// TwinCAT 3 PLC project TE1063
// ProgramVersion: 3.1.4024.0
// libraries:
//   CmpBitmapPool, * (System)
//   Tc2_Database, * (Beckhoff Automation GmbH)
//   Tc2_Math, * (Beckhoff Automation GmbH)
//   Tc2_MC2, * (Beckhoff Automation GmbH)
//   Tc2_SerialCom, * (Beckhoff Automation GmbH)
//   Tc2_Standard, * (Beckhoff Automation GmbH)
//   Tc2_System, * (Beckhoff Automation GmbH)
//   Tc2_TcpIp, * (Beckhoff Automation GmbH)
//   Tc2_Utilities, * (Beckhoff Automation GmbH)
//   Tc3_EventLogger, * (Beckhoff Automation GmbH)
//   Tc3_JsonXml, * (Beckhoff Automation GmbH)
//   Tc3_Module, * (Beckhoff Automation GmbH)
//   Base Interfaces,newest,System
//   VisuSymbols,3.5.10.0,System
// project tree:
//   DUTs/AlarmEventLogger/ E_Events.TcDUT, ST_GeneralAlarm.TcDUT, ST_PumpError.TcDUT (not stored), ST_ValveError.TcDUT
//   DUTs/AutoCycle/ E_MachineStates.TcDUT, E_PrimeSolventState.TcDUT, E_RecoveryState.TcDUT, E_WashingState.TcDUT
//   DUTs/Calibration/ E_LeakTestState.TcDUT, E_PState.TcDUT, E_StopState.TcDUT, E_CalibrationStatus.TcDUT, E_CalibStep.TcDUT, E_ScaleCmd.TcDUT, E_SolventType.TcDUT, ST_CalibrationData.TcDUT, ST_CalibrationInfo.TcDUT, ST_CalibrationPump.TcDUT, ST_CalibrationPumpResult.TcDUT, ST_DosingResults.TcDUT, ST_LinearPumpCalibration.TcDUT, ST_LinearPumpControllDB.TcDUT, ST_ReportInfo.TcDUT, ST_ScaleReply.TcDUT
//   DUTs/HMI/ E_IconState.TcDUT, E_MachineMode.TcDUT (not stored), ST_AX8101IOInfo.TcDUT, ST_AMI8000IOInfo.TcDUT, ST_HMIAnimation.TcDUT, ST_HMIDigInputs.TcDUT, ST_HMIDigOutputs.TcDUT, ST_HMIManual.TcDUT, ST_HMIParameters.TcDUT, ST_InfoPage.TcDUT, ST_EL7062IOInfo.TcDUT, ST_MotorsJog.TcDUT, ST_Reminders.TcDUT
//   DUTs/ifmLvlSensors/ E_LevelSensorID.TcDUT, ST_KQ1000_Data.TcDUT
//   DUTs/IO/ ST_AL1333.TcDUT, ST_AX8108.TcDUT, ST_EL1809.TcDUT, ST_EL2624.TcDUT, ST_EL2809.TcDUT, ST_EL3022.TcDUT (not stored), ST_EL3058.TcDUT, ST_EL6631.TcDUT, ST_EL6910.TcDUT, ST_EL7062.TcDUT, ST_EL7062A1.TcDUT, ST_EL7062A2.TcDUT, ST_EL7211.TcDUT, ST_EP9208.TcDUT
//   DUTs/ManualControl/ E_SolenoidSet.TcDUT, ST_MotorCommand.TcDUT, ST_PumpCommand.TcDUT, ST_ValveCommand.TcDUT
//   DUTs/MotionControl/ E_ActuatorState.TcDUT, E_MotorType.TcDUT, E_PumpDirection.TcDUT (not stored), E_PumpPath.TcDUT, ST_ActuatorStatus.TcDUT, ST_AxisReadStatus.TcDUT, ST_Motor.TcDUT, ST_SolenoidSet.TcDUT
//   DUTs/Recipe/ ST_HMI_OtherParamsRow.TcDUT, ST_HMI_SolventAndTimeRow.TcDUT, ST_HMI_VolumesRow.TcDUT, ST_Recipe.TcDUT, ST_RecipeFileInfo.TcDUT, ST_RecipeInfo.TcDUT, ST_RecipeOtherParams.TcDUT, ST_RecipeSolventAndTimes.TcDUT, ST_RecipeVolumes.TcDUT
//   DUTs/Report/ ST_CalibHeaderTest.TcDUT, E_ReportType.TcDUT, ST_CompleteMethodHeader.TcDUT, ST_LinearReport.TcDUT, ST_ReportListItem.TcDUT, ST_ReportListItem_Test.TcDUT, ST_ReportPostRun.TcDUT, ST_RunEvent.TcDUT, ST_SolventInfo.TcDUT, ST_SystemSettingsReport.TcDUT, ST_VolumeLine.TcDUT
//   DUTs/Safety/ ST_SafetyInputs.TcDUT, ST_SafetyOutputs.TcDUT
//   DUTs/Settings/ ST_CalibrationSettings.TcDUT, ST_LeakTestSettings.TcDUT, ST_PumpSettings.TcDUT, ST_SolventsSettings.TcDUT
//   DUTs/UserManagement/ E_UserGroup.TcDUT, ST_User.TcDUT, ST_UserStats.TcDUT
//   DUTs/Utility/ E_PowerAction.TcDUT, E_SeqState.TcDUT
//   GVLs/ GVL_Alarms.TcGVL, GVL_Calibration.TcGVL, GVL_Constant.TcGVL, GVL_HMI.TcGVL, GVL_IO.TcGVL, GVL_Reports.TcGVL, GVL_Retain.TcGVL, GVL_Settings.TcGVL, GVL_Motion.TcGVL, GVL_Recipe.TcGVL, GVL_Safety.TcGVL, GVL_UserManagement.TcGVL
//   / PlcTask.TcTTO, Task_Events.TcTTO, Task_HMI.TcTTO, Task_Services.TcTTO, Visualization Manager.TcVMO (not stored)
//   POUs/0. Main/ MAIN_Control.TcPOU, MAIN_Events.TcPOU, MAIN_HMI.TcPOU, MAIN_Services.TcPOU
//   POUs/2. AutoCycle/Hardware Control/ FB_SetSolenoid.TcPOU, FB_SolenoidControl.TcPOU
//   POUs/2. AutoCycle/ PRG_AutoCycle.TcPOU
//   POUs/2. AutoCycle/Stages/ FB_MeteringSolvent1.TcPOU, FB_PostRun.TcPOU, FB_PrimeSolvent.TcPOU, FB_AirFlowCheck.TcPOU, FB_DryingPhase.TcPOU, FB_InitChecks.TcPOU, FB_LeakTest.TcPOU, FB_RecoveryPhase.TcPOU, FB_SealStages.TcPOU, FB_WashingPhase.TcPOU
//   POUs/3. HMI/ PRG_HMIControl.TcPOU, PRG_SaveSolvents.TcPOU, PRG_SetModulestatus.TcPOU
//   POUs/5. Calibration/ FB_BuildCalReportJson.TcPOU, FB_CalibrationManager.TcPOU, FB_SaveCalibrationReport.TcPOU, FB_SaveCalReportToFile.TcPOU, FB_ScaleDevice.TcPOU, PRG_Calibration.TcPOU
//   POUs/6. Reports/ PRG_ReportsManager.TcPOU
//   POUs/7. EventsAndAlarms/ FB_AlarmHandler.TcPOU, FB_ErrorHandler.TcPOU, FB_EventHandler.TcPOU (not stored)
//   POUs/7. EventsAndAlarms/Marco/ POU_EventTest.TcPOU, POU_FaultHandler.TcPOU, PRG_MasterSystemTime.TcPOU
//   POUs/Functions/ F_AnyAxisMoving.TcPOU, F_GetPumpPath.TcPOU, F_GetValvePosition.TcPOU, F_JarName.TcPOU, F_MonthString.TcPOU (not stored), F_ParseWeight.TcPOU, F_REAL_TO_STRING_2DEC.TcPOU, F_ROUND_REAL.TcPOU, F_sec_to_time.TcPOU, F_TwoDigits.TcPOU (not stored), F_VolumeToSteps.TcPOU, F_VolumeToSteps_Path.TcPOU, F_SqlEscapeString.TcPOU
//   POUs/1. MachineControl/ PRG_ManualControl.TcPOU, PRG_MasterControl.TcPOU, PRG_SafetyHandle.TcPOU, PRG_StoppedState.TcPOU, PRG_SystemInit.TcPOU, PRG_SystemReady.TcPOU
//   POUs/Levels/ FB_KQ1000_Parser.TcPOU, FB_LevelSensors.TcPOU, PRG_LevelHandler.TcPOU
//   POUs/MARCO/DB/ DB_Edit_Method.TcPOU, DB_Load_CompleteMethod.TcPOU, DB_Query.TcPOU, GVL_DB.TcGVL, DB_Load_SysParameters.TcPOU, DB_Create_Calibration.TcPOU
//   POUs/MARCO/DB/STs/ E_DB_QUERY_STATE.TcTLEO, E_UserMgmtEventType.TcDUT, ST_CalibrationReportHeader.TcDUT, ST_CalibrationReportLine.TcDUT, ST_CalibrationReportListItem.TcDUT, ST_Data_CUL.TcDUT (not stored), ST_Data_PCR.TcDUT, ST_Data_UHR.TcDUT, ST_DB_Solvents.TcDUT, ST_LinearMotors.TcDUT, ST_ListMethod.TcDUT, ST_Parameters_MR.TcDUT, ST_CompleteMethod.TcDUT, ST_Parameters_PCR.TcDUT, ST_PostRunReport.TcDUT, ST_Results.TcDUT (not stored), ST_Solvents.TcDUT, ST_SysParameters.TcDUT, ST_UserMgmtHistoryEvent.TcDUT, ST_VolumeData.TcDUT
//   POUs/MARCO/OLD/ GVL_Marco.TcGVL, POU_Master_Calib.TcPOU, POU_Master_Calib_1.TcPOU, POU_Master_Calib_2.TcPOU, POU_Motion.TcPOU (not stored)
//   POUs/Utilities/ FB_Blink.TcPOU (not stored), FB_DosingTest.TcPOU, FB_EventLog.TcPOU (not stored), FB_SensorScaling.TcPOU, FB_TCPClient.TcPOU, PRG_PowerManagement.TcPOU (not stored), PRG_RetainValveAngles.TcPOU (not stored), PRG_ShutdownPLC.TcPOU (not stored), PRG_SystemInfo.TcPOU (not stored), PRG_TowerAlarmLamps.TcPOU, PRG_UpdateVariablesMoving.TcPOU, PRG_UserManagementHistory.TcPOU, PRG_ValvePositionRecovery.TcPOU (not stored), PRG_ValveTest.TcPOU
//   POUs/MotionControl/ FB_AllPumpsController.TcPOU, FB_MotorWrapper.TcPOU, IF_Actuator.TcIO, PRG_AxisAssignment.TcPOU
//   POUs/4. RecipeHandle/ FB_DeleteRecipe.TcPOU, FB_ListRecipeFiles.TcPOU, FB_LoadRecipe.TcPOU, FB_RecipeHeaderHandler.TcPOU, FB_SaveRecipe.TcPOU, PRG_RecipeManager.TcPOU
//   VISUs/ GlobalTextList.TcGTLO, Visualization.TcVIS
// real-time tasks:
//   TASK Task_Control: cycle T#10ms, priority 10, ADS port 350
//   TASK Task_HMI: cycle T#100000us, priority 12, ADS port 351
//   TASK Task_Events: cycle T#250ms, priority 14, ADS port 352
//   TASK Task_Services: cycle T#1000ms, priority 16, ADS port 353
// motion (NC):
//   TASK NC-Task 1 SAF: cycle T#2ms, priority 4, ADS port 501
//   TASK NC-Task 1 SVB: cycle T#2ms, priority 6, ADS port 511
//   AXIS M1 Motor - SR Vertical (id 28)
//     General: UnitFlags=#x00000001
//     Dynamic: Acceleration=58.278, Deceleration=58.278, Jerk=174.834
//     Velo: RefSearch=0.38852, RefSync=0.38852, SlowManual=1.25, FastManual=7.5, Fast=38.852, Maximum=38.852
//     OtherSettings: AllowMotionCmdToSlave=true
//     encoder EncType=19
//       EncPara: ScaleFactorNumerator=25, ScaleFactorDenominator=20971520, MaxCount=#xffffffff
//     drive DrvType=16
//       DrvPara: MaxCount=#xffffffff, DriveControlDWord=#x00020100
//         Analog: VeloReferenz=42.7372, VeloScale=71.5255737304688, TorqueSetpointScale=10, ScaleFactorActTorque=0.1
//         TimeComp: TaskDelayCycles=1
//     controller CtrType=1
//       CtrPara: PriorControlFactor=1
//         Observer: BandWidth=20
//   AXIS M2 Motor - SC Vertical (id 6)
//     Dynamic: AccelerationMaximum=15, DecelerationMaximum=15, Acceleration=15, Deceleration=15, Jerk=2457.738
//     Velo: RefSearch=5.46164, RefSync=5.46164, SlowManual=2, FastManual=6, Fast=546.164, Maximum=546.164
//     OtherSettings: AllowMotionCmdToSlave=true, PulseDistancePos=1, PulseDistanceNeg=1
//     encoder EncType=19
//       EncPara: ScaleFactorNumerator=10, ScaleFactorDenominator=1048576, MaxCount=#xffffffff
//         TimeComp: TimeCompMode=1, EncDelayCycles=4
//     drive DrvType=16
//       DrvPara: MaxCount=#xffffffff, DriveControlDWord=#x00020100
//         Analog: VeloReferenz=600.7804, VeloScale=32, TorqueSetpointScale=10, ScaleFactorActTorque=0.1
//         TimeComp: TaskDelayCycles=1
//     controller CtrType=1
//       CtrPara: PriorControlFactor=1
//         Observer: BandWidth=20
//   AXIS M3 Motor - SC Horizontal (id 7)
//     Dynamic: Acceleration=819.246, Deceleration=819.246, Jerk=2457.738
//     Velo: RefSearch=5.46164, RefSync=5.46164, SlowManual=6, FastManual=12, Fast=546.164, Maximum=546.164
//     OtherSettings: AllowMotionCmdToSlave=true, PulseDistancePos=2, PulseDistanceNeg=2
//     encoder EncType=19
//       EncPara: ScaleFactorNumerator=10, ScaleFactorDenominator=1048576, MaxCount=#xffffffff
//     drive DrvType=16
//       DrvPara: MaxCount=#xffffffff, DriveControlDWord=#x00020100
//         Analog: VeloReferenz=600.7804, VeloScale=32, TorqueSetpointScale=10, ScaleFactorActTorque=0.1
//         TimeComp: TaskDelayCycles=1
//     controller CtrType=1
//       CtrPara: PriorControlFactor=1
//         Observer: BandWidth=20
//   AXIS M4 Motor - Valve 1 (id 1)
//     General: UnitName=°
//     Dynamic: Acceleration=15000, Deceleration=15000, Jerk=88478.5
//     Velo: RefSearch=196.61898, RefSync=196.61898, SlowManual=300, FastManual=1000, Fast=19661.898, Maximum=19661.9
//     OtherSettings: AllowMotionCmdToSlave=true, PulseDistancePos=1, PulseDistanceNeg=1
//     encoder EncType=19
//       EncPara: ScaleFactorNumerator=360, ScaleFactorDenominator=1048576, Offset=959.925842285156, MaxCount=#xffffffff, ReferenceSystem=4
//         SoftEndMaxControl: Range=7200
//     drive DrvType=16
//       DrvPara: MaxCount=#xffffffff, DriveControlDWord=#x00020100
//         Analog: VeloReferenz=21628.0878, VeloScale=32, TorqueSetpointScale=10, ScaleFactorActTorque=0.1
//         TimeComp: TaskDelayCycles=1
//     controller CtrType=1
//       CtrPara: PriorControlFactor=1
//         PosDiffControl: Range=90
//         Observer: BandWidth=20
//   AXIS M5 Motor - Valve 2 (id 2)
//     General: UnitName=°
//     Dynamic: Acceleration=15000, Deceleration=15000, Jerk=88478.5
//     Velo: RefSearch=196.61898, RefSync=196.61898, SlowManual=300, FastManual=1000, Fast=19661.898, Maximum=19661.9
//     OtherSettings: AllowMotionCmdToSlave=true, PulseDistancePos=1, PulseDistanceNeg=1
//     encoder EncType=19
//       EncPara: ScaleFactorNumerator=360, ScaleFactorDenominator=1048576, MaxCount=#xffffffff, ReferenceSystem=4
//     drive DrvType=16
//       DrvPara: MaxCount=#xffffffff, DriveControlDWord=#x00020100
//         Analog: VeloReferenz=21628.0878, VeloScale=32, TorqueSetpointScale=10, ScaleFactorActTorque=0.1
//         TimeComp: TaskDelayCycles=1
//     controller CtrType=1
//       CtrPara: PriorControlFactor=1
//         PosDiffControl: Range=90
//         Observer: BandWidth=20
//   AXIS M6 Motor - Valve 3 (id 29)
//     General: UnitName=°
//     Dynamic: Acceleration=15000, Deceleration=15000, Jerk=88478.5
//     Velo: RefSearch=196.61898, RefSync=196.61898, SlowManual=300, FastManual=1000, Fast=19661.898, Maximum=19661.9
//     OtherSettings: AllowMotionCmdToSlave=true, PulseDistancePos=1, PulseDistanceNeg=1
//     encoder EncType=19
//       EncPara: ScaleFactorNumerator=360, ScaleFactorDenominator=1048576, MaxCount=#xffffffff, ReferenceSystem=4
//     drive DrvType=16
//       DrvPara: MaxCount=#xffffffff, DriveControlDWord=#x00020100
//         Analog: VeloReferenz=21628.0878, VeloScale=32, TorqueSetpointScale=10, ScaleFactorActTorque=0.1
//         TimeComp: TaskDelayCycles=1
//     controller CtrType=1
//       CtrPara: PriorControlFactor=1
//         PosDiffControl: Range=90
//         Observer: BandWidth=20
//   AXIS M7 Motor - Valve 4 (id 4)
//     General: UnitName=°
//     Dynamic: Acceleration=15000, Deceleration=15000, Jerk=88478.5
//     Velo: RefSearch=196.61898, RefSync=196.61898, SlowManual=300, FastManual=1000, Fast=19661.898, Maximum=19661.9
//     OtherSettings: AllowMotionCmdToSlave=true, PulseDistancePos=1, PulseDistanceNeg=1
//     encoder EncType=19
//       EncPara: ScaleFactorNumerator=360, ScaleFactorDenominator=1048576, MaxCount=#xffffffff, ReferenceSystem=4
//     drive DrvType=16
//       DrvPara: MaxCount=#xffffffff, DriveControlDWord=#x00020100
//         Analog: VeloReferenz=21628.0878, VeloScale=32, TorqueSetpointScale=10, ScaleFactorActTorque=0.1
//         TimeComp: TaskDelayCycles=1
//     controller CtrType=1
//       CtrPara: PriorControlFactor=1
//         PosDiffControl: Range=90
//         Observer: BandWidth=20
//   AXIS M8 Motor - Valve 5 (id 5)
//     General: UnitName=°
//     Dynamic: Acceleration=15000, Deceleration=15000, Jerk=88478.541
//     Velo: RefSearch=196.61898, RefSync=196.61898, SlowManual=300, FastManual=1000, Fast=19661.898, Maximum=19661.898
//     OtherSettings: AllowMotionCmdToSlave=true, PulseDistancePos=1, PulseDistanceNeg=1
//     encoder EncType=19
//       EncPara: ScaleFactorNumerator=360, ScaleFactorDenominator=1048576, MaxCount=#xffffffff, ReferenceSystem=4
//     drive DrvType=16
//       DrvPara: MaxCount=#xffffffff, DriveControlDWord=#x00020100
//         Analog: VeloReferenz=21628.0878, VeloScale=32, TorqueSetpointScale=10, ScaleFactorActTorque=0.1
//         TimeComp: TaskDelayCycles=1
//     controller CtrType=1
//       CtrPara: PriorControlFactor=1
//         PosDiffControl: Range=90
//         Observer: BandWidth=20
//   AXIS Pump 1 - Linear (id 8)
//     Dynamic: Acceleration=7200, Deceleration=7200, Jerk=21600
//     Velo: RefSearch=48, RefSync=48, SlowManual=50, FastManual=100, Fast=4800, Maximum=4800
//     OtherSettings: AllowMotionCmdToSlave=true, PulseDistancePos=1, PulseDistanceNeg=1
//     encoder EncType=19
//       EncPara: ScaleFactorNumerator=200, ScaleFactorDenominator=1048576, MaxCount=#xffffffff
//         SoftEndMinControl: Range=-4500
//         SoftEndMaxControl: Range=500
//     drive DrvType=16
//       DrvPara: MaxCount=#xffffffff, DriveControlDWord=#x00020100
//         Analog: VeloReferenz=5280, VeloScale=32, TorqueSetpointScale=10, ScaleFactorActTorque=0.1
//         TimeComp: TaskDelayCycles=1
//     controller CtrType=1
//       CtrPara: PriorControlFactor=1
//         Observer: BandWidth=20
//   AXIS Pump 1 - Rotary (id 9)
//     General: UnitName=°
//     Dynamic: AccelerationMaximum=1500, DecelerationMaximum=1500, Jerk=21793.7205
//     Velo: RefSearch=48.43049, RefSync=48.43049, SlowManual=242.15245, FastManual=1452.9147, Fast=4843.049, Maximum=6000
//     OtherSettings: AllowMotionCmdToSlave=true
//     encoder EncType=19
//       EncPara: ScaleFactorNumerator=360, ScaleFactorDenominator=1048576, MaxCount=#xffffffff
//         Inc: RefSyncInverse=false
//     drive DrvType=16
//       DrvPara: MaxCount=#xffffffff, DriveControlDWord=#x00020100
//         Analog: VeloReferenz=5500, VeloScale=32, TorqueSetpointScale=10, ScaleFactorActTorque=0.1
//         TimeComp: TaskDelayCycles=1
//     controller CtrType=2
//       CtrPara: PriorControlFactor=1
//         PosDiffControl: Range=200
//         Observer: BandWidth=20
//   AXIS Pump 2 - Linear (id 10)
//     Dynamic: Acceleration=7200, Deceleration=7200, Jerk=21600
//     Velo: RefSearch=48, RefSync=48, SlowManual=50, FastManual=100, Fast=4800, Maximum=4800
//     OtherSettings: AllowMotionCmdToSlave=true, PulseDistancePos=1, PulseDistanceNeg=1
//     encoder EncType=19
//       EncPara: ScaleFactorNumerator=200, ScaleFactorDenominator=1048576, MaxCount=#xffffffff
//         SoftEndMinControl: Range=-4500
//         SoftEndMaxControl: Range=500
//     drive DrvType=16
//       DrvPara: MaxCount=#xffffffff, DriveControlDWord=#x00020100
//         Analog: VeloReferenz=5280, VeloScale=32, TorqueSetpointScale=10, ScaleFactorActTorque=0.1
//         TimeComp: TaskDelayCycles=1
//     controller CtrType=1
//       CtrPara: PriorControlFactor=1
//         Observer: BandWidth=20
//   AXIS Pump 2 - Rotary (id 11)
//     General: UnitName=°
//     Dynamic: Acceleration=7264.5735, Deceleration=7264.5735, Jerk=21793.7205
//     Velo: RefSearch=48.43049, RefSync=48.43049, SlowManual=500, FastManual=3600, Fast=4843.049, Maximum=4843.049
//     OtherSettings: AllowMotionCmdToSlave=true
//     encoder EncType=19
//       EncPara: ScaleFactorNumerator=360, ScaleFactorDenominator=1048576, MaxCount=#xffffffff
//     drive DrvType=16
//       DrvPara: MaxCount=#xffffffff, DriveControlDWord=#x00020100
//         Analog: VeloReferenz=5327.3539, TorqueSetpointScale=10, ScaleFactorActTorque=0.1
//         TimeComp: TaskDelayCycles=1
//     controller CtrType=1
//       CtrPara: PriorControlFactor=1
//         Observer: BandWidth=20
//   AXIS Pump 3 - Linear (id 12)
//     Dynamic: Acceleration=7200, Deceleration=7200, Jerk=21600
//     Velo: RefSearch=48, RefSync=48, SlowManual=50, FastManual=100, Fast=4800, Maximum=4800
//     OtherSettings: AllowMotionCmdToSlave=true, PulseDistancePos=1, PulseDistanceNeg=1
//     encoder EncType=19
//       EncPara: ScaleFactorNumerator=200, ScaleFactorDenominator=1048576, MaxCount=#xffffffff
//         SoftEndMinControl: Range=-4500
//         SoftEndMaxControl: Range=500
//     drive DrvType=16
//       DrvPara: MaxCount=#xffffffff, DriveControlDWord=#x00020100
//         Analog: VeloReferenz=5280, VeloScale=32, TorqueSetpointScale=10, ScaleFactorActTorque=0.1
//         TimeComp: TaskDelayCycles=1
//     controller CtrType=1
//       CtrPara: PriorControlFactor=1
//         Observer: BandWidth=20
//   AXIS Pump 3 - Rotary (id 13)
//     General: UnitName=°
//     Dynamic: Acceleration=7264.57, Deceleration=7264.57, Jerk=21793.7
//     Velo: RefSearch=48.43049, RefSync=48.43049, SlowManual=500, FastManual=3600, Fast=4843.049, Maximum=4843.05
//     OtherSettings: AllowMotionCmdToSlave=true
//     encoder EncType=19
//       EncPara: ScaleFactorNumerator=360, ScaleFactorDenominator=1048576, MaxCount=#xffffffff
//         Inc: RefSyncInverse=false
//     drive DrvType=16
//       DrvPara: MaxCount=#xffffffff, DriveControlDWord=#x00020100
//         Analog: VeloReferenz=5327.3539, VeloScale=32, TorqueSetpointScale=10, ScaleFactorActTorque=0.1
//         TimeComp: TaskDelayCycles=1
//     controller CtrType=1
//       CtrPara: PriorControlFactor=1
//         PosDiffControl: Enable=false
//         Observer: BandWidth=20
//   AXIS Pump 4 - Linear (id 14)
//     Dynamic: Acceleration=7200, Deceleration=7200, Jerk=21600
//     Velo: RefSearch=48, RefSync=48, SlowManual=50, FastManual=100, Fast=4800, Maximum=4800
//     OtherSettings: AllowMotionCmdToSlave=true, PulseDistancePos=1, PulseDistanceNeg=1
//     encoder EncType=19
//       EncPara: ScaleFactorNumerator=200, ScaleFactorDenominator=1048576, MaxCount=#xffffffff
//         SoftEndMinControl: Range=-4500
//         SoftEndMaxControl: Range=500
//     drive DrvType=16
//       DrvPara: MaxCount=#xffffffff, DriveControlDWord=#x00020100
//         Analog: VeloReferenz=5280, VeloScale=32, TorqueSetpointScale=10, ScaleFactorActTorque=0.1
//         TimeComp: TaskDelayCycles=1
//     controller CtrType=1
//       CtrPara: PriorControlFactor=1
//         Observer: BandWidth=20
//   AXIS Pump 4 - Rotary (id 15)
//     General: UnitName=°
//     Dynamic: AccelerationMaximum=100, DecelerationMaximum=100, Acceleration=100, Deceleration=100, Jerk=21793.7205
//     Velo: RefSearch=48.43049, RefSync=48.43049, SlowManual=242.15245, FastManual=1452.9147, Fast=4843.049, Maximum=4843.049
//     OtherSettings: AllowMotionCmdToSlave=true
//     encoder EncType=19
//       EncPara: ScaleFactorNumerator=360, ScaleFactorDenominator=1048576, MaxCount=#xffffffff
//     drive DrvType=16
//       DrvPara: MaxCount=#xffffffff, DriveControlDWord=#x00020100
//         Analog: VeloReferenz=5327.3539, TorqueSetpointScale=10, ScaleFactorActTorque=0.1
//         TimeComp: TaskDelayCycles=1
//     controller CtrType=1
//       CtrPara: PriorControlFactor=1
//         Observer: BandWidth=20
//   AXIS Pump 5 - Linear (id 16)
//     Dynamic: Acceleration=7200, Deceleration=7200, Jerk=21600
//     Velo: RefSearch=48, RefSync=48, SlowManual=50, FastManual=100, Fast=4800, Maximum=4800
//     OtherSettings: AllowMotionCmdToSlave=true, PulseDistancePos=1, PulseDistanceNeg=1
//     encoder EncType=19
//       EncPara: ScaleFactorNumerator=200, ScaleFactorDenominator=1048576, MaxCount=#xffffffff
//         SoftEndMinControl: Range=-4500
//         SoftEndMaxControl: Range=500
//     drive DrvType=16
//       DrvPara: MaxCount=#xffffffff, DriveControlDWord=#x00020100
//         Analog: VeloReferenz=5280, VeloScale=32, TorqueSetpointScale=10, ScaleFactorActTorque=0.1
//         TimeComp: TaskDelayCycles=1
//     controller CtrType=1
//       CtrPara: PriorControlFactor=1
//         Observer: BandWidth=20
//   AXIS Pump 5 - Rotary (id 17)
//     General: UnitName=°
//     Dynamic: Acceleration=7264.57, Deceleration=7264.57, Jerk=21793.7
//     Velo: RefSearch=48.43049, RefSync=48.43049, SlowManual=500, FastManual=3600, Fast=4843.049, Maximum=4843.05
//     OtherSettings: AllowMotionCmdToSlave=true
//     encoder EncType=19
//       EncPara: ScaleFactorNumerator=360, ScaleFactorDenominator=1048576, MaxCount=#xffffffff
//     drive DrvType=16
//       DrvPara: MaxCount=#xffffffff, DriveControlDWord=#x00020100
//         Analog: VeloReferenz=5327.3539, VeloScale=32, TorqueSetpointScale=10, ScaleFactorActTorque=0.1
//         TimeComp: TaskDelayCycles=1
//     controller CtrType=1
//       CtrPara: PriorControlFactor=1
//         Observer: BandWidth=20
//   AXIS Pump 6 - Linear (id 18)
//     Dynamic: Acceleration=7200, Deceleration=7200, Jerk=21600
//     Velo: RefSearch=48, RefSync=48, SlowManual=50, FastManual=100, Fast=4800, Maximum=4800
//     OtherSettings: AllowMotionCmdToSlave=true, PulseDistancePos=1, PulseDistanceNeg=1
//     encoder EncType=19
//       EncPara: ScaleFactorNumerator=200, ScaleFactorDenominator=1048576, MaxCount=#xffffffff
//         SoftEndMinControl: Range=-4500
//         SoftEndMaxControl: Range=500
//     drive DrvType=16
//       DrvPara: MaxCount=#xffffffff, DriveControlDWord=#x00020100
//         Analog: VeloReferenz=5280, VeloScale=32, TorqueSetpointScale=10, ScaleFactorActTorque=0.1
//         TimeComp: TaskDelayCycles=1
//     controller CtrType=1
//       CtrPara: PriorControlFactor=1
//         Observer: BandWidth=20
//   AXIS Pump 6 - Rotary (id 19)
//     General: UnitName=°
//     Dynamic: Acceleration=7264.57, Deceleration=7264.57, Jerk=21793.7
//     Velo: RefSearch=48.43049, RefSync=48.43049, SlowManual=500, FastManual=3600, Fast=4843.049, Maximum=4843.05
//     OtherSettings: AllowMotionCmdToSlave=true
//     encoder EncType=19
//       EncPara: ScaleFactorNumerator=360, ScaleFactorDenominator=1048576, MaxCount=#xffffffff
//     drive DrvType=16
//       DrvPara: MaxCount=#xffffffff, DriveControlDWord=#x00020100
//         Analog: VeloReferenz=5327.3539, VeloScale=32, TorqueSetpointScale=10, ScaleFactorActTorque=0.1
//         TimeComp: TaskDelayCycles=1
//     controller CtrType=1
//       CtrPara: PriorControlFactor=1
//         Observer: BandWidth=20
//   AXIS Pump 7 - Linear (id 20)
//     Dynamic: Acceleration=7200, Deceleration=7200, Jerk=21600
//     Velo: RefSearch=48, RefSync=48, SlowManual=50, FastManual=100, Fast=4800, Maximum=4800
//     OtherSettings: AllowMotionCmdToSlave=true, PulseDistancePos=1, PulseDistanceNeg=1
//     encoder EncType=19
//       EncPara: ScaleFactorNumerator=200, ScaleFactorDenominator=1048576, MaxCount=#xffffffff
//         SoftEndMinControl: Range=-4500
//         SoftEndMaxControl: Range=500
//     drive DrvType=16
//       DrvPara: MaxCount=#xffffffff, DriveControlDWord=#x00020100
//         Analog: VeloReferenz=5280, VeloScale=32, TorqueSetpointScale=10, ScaleFactorActTorque=0.1
//         TimeComp: TaskDelayCycles=1
//     controller CtrType=1
//       CtrPara: PriorControlFactor=1
//         Observer: BandWidth=20
//   AXIS Pump 7 - Rotary (id 21)
//     General: UnitName=°
//     Dynamic: Acceleration=7264.5735, Deceleration=7264.5735, Jerk=21793.7205
//     Velo: RefSearch=48.43049, RefSync=48.43049, SlowManual=500, FastManual=3600, Fast=4843.049, Maximum=4843.049
//     OtherSettings: AllowMotionCmdToSlave=true
//     encoder EncType=19
//       EncPara: ScaleFactorNumerator=360, ScaleFactorDenominator=1048576, MaxCount=#xffffffff
//     drive DrvType=16
//       DrvPara: MaxCount=#xffffffff, DriveControlDWord=#x00020100
//         Analog: VeloReferenz=5327.3539, VeloScale=32, TorqueSetpointScale=10, ScaleFactorActTorque=0.1
//         TimeComp: TaskDelayCycles=1
//     controller CtrType=1
//       CtrPara: PriorControlFactor=1
//         Observer: BandWidth=20
//   AXIS Pump 8 - Linear (id 22)
//     Dynamic: Acceleration=7200, Deceleration=7200, Jerk=21600
//     Velo: RefSearch=48, RefSync=48, SlowManual=50, FastManual=100, Fast=4800, Maximum=4800
//     OtherSettings: AllowMotionCmdToSlave=true, PulseDistancePos=1, PulseDistanceNeg=1
//     encoder EncType=19
//       EncPara: ScaleFactorNumerator=200, ScaleFactorDenominator=1048576, MaxCount=#xffffffff
//         SoftEndMinControl: Range=-4500
//         SoftEndMaxControl: Range=500
//     drive DrvType=16
//       DrvPara: MaxCount=#xffffffff, DriveControlDWord=#x00020100
//         Analog: VeloReferenz=5280, VeloScale=32, TorqueSetpointScale=10, ScaleFactorActTorque=0.1
//         TimeComp: TaskDelayCycles=1
//     controller CtrType=1
//       CtrPara: PriorControlFactor=1
//         Observer: BandWidth=20
//   AXIS Pump 8 - Rotary (id 23)
//     General: UnitName=°
//     Dynamic: Acceleration=7264.5735, Deceleration=7264.5735, Jerk=21793.7205
//     Velo: RefSearch=48.43049, RefSync=48.43049, SlowManual=500, FastManual=3600, Fast=4843.049, Maximum=4843.049
//     OtherSettings: AllowMotionCmdToSlave=true
//     encoder EncType=19
//       EncPara: ScaleFactorNumerator=360, ScaleFactorDenominator=1048576, MaxCount=#xffffffff
//     drive DrvType=16
//       DrvPara: MaxCount=#xffffffff, DriveControlDWord=#x00020100
//         Analog: VeloReferenz=5327.3539, VeloScale=32, TorqueSetpointScale=10, ScaleFactorActTorque=0.1
//         TimeComp: TaskDelayCycles=1
//     controller CtrType=1
//       CtrPara: PriorControlFactor=1
//         Observer: BandWidth=20
//   AXIS Pump 9 - Linear (id 24)
//     Dynamic: Acceleration=7200, Deceleration=7200, Jerk=21600
//     Velo: RefSearch=48, RefSync=48, SlowManual=50, FastManual=100, Fast=4800, Maximum=4800
//     OtherSettings: AllowMotionCmdToSlave=true, PulseDistancePos=1, PulseDistanceNeg=1
//     encoder EncType=19
//       EncPara: ScaleFactorNumerator=200, ScaleFactorDenominator=1048576, MaxCount=#xffffffff
//         SoftEndMinControl: Range=-4500
//         SoftEndMaxControl: Range=500
//     drive DrvType=16
//       DrvPara: MaxCount=#xffffffff, DriveControlDWord=#x00020100
//         Analog: VeloReferenz=5280, VeloScale=32, TorqueSetpointScale=10, ScaleFactorActTorque=0.1
//         TimeComp: TaskDelayCycles=1
//     controller CtrType=1
//       CtrPara: PriorControlFactor=1
//         Observer: BandWidth=20
//   AXIS Pump 9 - Rotary (id 25)
//     General: UnitName=°
//     Dynamic: Acceleration=7264.5735, Deceleration=7264.5735, Jerk=21793.7205
//     Velo: RefSearch=48.43049, RefSync=48.43049, SlowManual=500, FastManual=3600, Fast=4843.049, Maximum=4843.049
//     OtherSettings: AllowMotionCmdToSlave=true
//     encoder EncType=19
//       EncPara: ScaleFactorNumerator=360, ScaleFactorDenominator=1048576, MaxCount=#xffffffff
//     drive DrvType=16
//       DrvPara: MaxCount=#xffffffff, DriveControlDWord=#x00020100
//         Analog: VeloReferenz=5327.3539, VeloScale=32, TorqueSetpointScale=10, ScaleFactorActTorque=0.1
//         TimeComp: TaskDelayCycles=1
//     controller CtrType=1
//       CtrPara: PriorControlFactor=1
//         Observer: BandWidth=20
//   AXIS Pump 10 - Linear (id 26)
//     Dynamic: Acceleration=7200, Deceleration=7200, Jerk=21600
//     Velo: RefSearch=48, RefSync=48, SlowManual=50, FastManual=100, Fast=4800, Maximum=4800
//     OtherSettings: AllowMotionCmdToSlave=true, PulseDistancePos=1, PulseDistanceNeg=1
//     encoder EncType=19
//       EncPara: ScaleFactorNumerator=200, ScaleFactorDenominator=1048576, MaxCount=#xffffffff
//         SoftEndMinControl: Range=-4500
//         SoftEndMaxControl: Range=500
//     drive DrvType=16
//       DrvPara: MaxCount=#xffffffff, DriveControlDWord=#x00020100
//         Analog: VeloReferenz=5280, VeloScale=32, TorqueSetpointScale=10, ScaleFactorActTorque=0.1
//         TimeComp: TaskDelayCycles=1
//     controller CtrType=1
//       CtrPara: PriorControlFactor=1
//         Observer: BandWidth=20
//   AXIS Pump 10 - Rotary (id 27)
//     General: UnitName=°
//     Dynamic: Acceleration=7264.5735, Deceleration=7264.5735, Jerk=21793.7205
//     Velo: RefSearch=48.43049, RefSync=48.43049, SlowManual=500, FastManual=3600, Fast=4843.049, Maximum=4843.049
//     OtherSettings: AllowMotionCmdToSlave=true
//     encoder EncType=19
//       EncPara: ScaleFactorNumerator=360, ScaleFactorDenominator=1048576, MaxCount=#xffffffff
//     drive DrvType=16
//       DrvPara: MaxCount=#xffffffff, DriveControlDWord=#x00020100
//         Analog: VeloReferenz=5327.3539, VeloScale=32, TorqueSetpointScale=10, ScaleFactorActTorque=0.1
//         TimeComp: TaskDelayCycles=1
//     controller CtrType=1
//       CtrPara: PriorControlFactor=1
//         Observer: BandWidth=20
// I/O:
//   DEVICE Device 1 (Virtual-Ethernet) (disabled)
//   DEVICE Device 4 (EtherCAT Automation Protocol) (disabled), AmsNetId 192.168.0.162.5.1
//   DEVICE Device 6 (EtherCAT), AmsNetId 192.168.0.162.7.1
//     Box 8 (AMI8000-0100) [AMI8000-0100 Servo motor 48 V DC, TwinSAFE]
//       modules: Module 1 (SAFETY)
//       startup 32785:21 := 0E01 // DRV Motor Settings / Commutation offset
//       startup 28688:11 := 640F // DRV Outputs / Torque limitation
//       startup 32784:19 := 9D00 // DRV Amplifier Settings / Current loop proportional gain
//       startup 32784:18 := 1100 // DRV Amplifier Settings / Current loop integral time
//       startup 32784:21 := 5F000000 // DRV Amplifier Settings / Velocity loop proportional gain
//       startup 32784:20 := 96000000 // DRV Amplifier Settings / Velocity loop integral time
//       startup 32768:21 := 64 // FB Settings / Observer feed-forward
//     Box 9 (AMI8000-0100) [AMI8000-0100 Servo motor 48 V DC, TwinSAFE]
//       modules: Module 1 (SAFETY)
//       startup 32785:21 := 0E01 // DRV Motor Settings / Commutation offset
//       startup 28688:11 := 640F // DRV Outputs / Torque limitation
//       startup 32784:19 := 9D00 // DRV Amplifier Settings / Current loop proportional gain
//       startup 32784:18 := 1100 // DRV Amplifier Settings / Current loop integral time
//       startup 32784:21 := 5F000000 // DRV Amplifier Settings / Velocity loop proportional gain
//       startup 32784:20 := 96000000 // DRV Amplifier Settings / Velocity loop integral time
//       startup 32768:21 := 64 // FB Settings / Observer feed-forward
//     Box 10 (AMI8000-0100) [AMI8000-0100 Servo motor 48 V DC, TwinSAFE]
//       modules: Module 1 (SAFETY)
//       startup 32785:21 := 0E01 // DRV Motor Settings / Commutation offset
//       startup 28688:11 := 640F // DRV Outputs / Torque limitation
//       startup 32784:19 := 9D00 // DRV Amplifier Settings / Current loop proportional gain
//       startup 32784:18 := 1100 // DRV Amplifier Settings / Current loop integral time
//       startup 32784:21 := 5F000000 // DRV Amplifier Settings / Velocity loop proportional gain
//       startup 32784:20 := 96000000 // DRV Amplifier Settings / Velocity loop integral time
//       startup 32768:21 := 64 // FB Settings / Observer feed-forward
//     Box 11 (AMI8000-0100) [AMI8000-0100 Servo motor 48 V DC, TwinSAFE]
//       modules: Module 1 (SAFETY)
//       startup 32785:21 := 0E01 // DRV Motor Settings / Commutation offset
//       startup 28688:11 := 640F // DRV Outputs / Torque limitation
//       startup 32784:19 := 9D00 // DRV Amplifier Settings / Current loop proportional gain
//       startup 32784:18 := 1100 // DRV Amplifier Settings / Current loop integral time
//       startup 32784:21 := 5F000000 // DRV Amplifier Settings / Velocity loop proportional gain
//       startup 32784:20 := 96000000 // DRV Amplifier Settings / Velocity loop integral time
//       startup 32768:21 := 64 // FB Settings / Observer feed-forward
//     Box 12 (AMI8000-0100) [AMI8000-0100 Servo motor 48 V DC, TwinSAFE]
//       modules: Module 1 (SAFETY)
//       startup 32785:21 := 0E01 // DRV Motor Settings / Commutation offset
//       startup 28688:11 := 640F // DRV Outputs / Torque limitation
//       startup 32784:19 := 9D00 // DRV Amplifier Settings / Current loop proportional gain
//       startup 32784:18 := 1100 // DRV Amplifier Settings / Current loop integral time
//       startup 32784:21 := 5F000000 // DRV Amplifier Settings / Velocity loop proportional gain
//       startup 32784:20 := 96000000 // DRV Amplifier Settings / Velocity loop integral time
//       startup 32768:21 := 64 // FB Settings / Observer feed-forward
//   DEVICE Device 3 (EtherCAT), AmsNetId 192.168.0.162.4.1
//     Term 1 (EK1100) [EK1100 EtherCAT Coupler (2A E-Bus)]
//       Term 2 (EL6070-0033) [EL6070-0033 1Ch. Licence key terminal, individual licences]
//       Term 3 (EL6910) [EL6910, TwinSAFE PLC]
//       Term 4 (EL1918) [EL1918, 8Ch. Safety Input 24V, TwinSAFE]
//         modules: Module 1 (FSOE), Module 2 (FSLOGIC)
//       Term 5 (EL1918) [EL1918, 8Ch. Safety Input 24V, TwinSAFE]
//         modules: Module 1 (FSOE), Module 2 (FSLOGIC)
//       Term 6 (EL1918) [EL1918, 8Ch. Safety Input 24V, TwinSAFE]
//         modules: Module 1 (FSOE), Module 2 (FSLOGIC)
//       Term 7 (EL2904) [EL2904, 4 Ch. Safety Output 24V, 0.5A, TwinSAFE]
//         modules: Module 1 (FSOES), Module 2 (DO)
//       Term 8 (EL2904) [EL2904, 4 Ch. Safety Output 24V, 0.5A, TwinSAFE]
//         modules: Module 1 (FSOES), Module 2 (DO)
//       Term 9 (EL1809) [EL1809 16Ch. Dig. Input 24V, 3ms]
//       Term 10 (EL2809-0015) [EL2809-0015 16Ch. Dig. Output 24V DC, 0.35A, not short-circuit proof]
//       Term 11 (EL2624) [EL2624 4Ch. Relay Output, NO (125V AC / 30V DC)]
//       Term 12 (EL9410) [EL9410 E-Bus Power Supplier  (Diagnostics)]
//       Term 13 (EL3058) [EL3058 8Ch. Ana. Input 4-20mA]
//       Term 14 (EL9576) [EL9576 Brake chopper terminal]
//       Term 15 (EL7211-9014) [EL7211-9014 1Ch. MDP742 Servo motor output stage with OCT (50V, 4.5A RMS) and STO input]
//         startup 32785:21 := 0E01 // DRV Motor Settings / Commutation offset
//         startup 32786:19 := 0000 // DRV Brake Settings / Emergency application timeout
//         startup 32784:51 := 0A00 // DRV Amplifier Settings / Stand still window
//         startup 32785:27 := D30C0000 // DRV Motor Settings / Motor speed limitation
//         startup 28688:11 := D007 // DRV Outputs / Torque limitation
//         startup 32784:19 := 4C01 // DRV Amplifier Settings / Current loop proportional gain
//         startup 32784:18 := 0500 // DRV Amplifier Settings / Current loop integral time
//         startup 32784:21 := 95000000 // DRV Amplifier Settings / Velocity loop proportional gain
//         startup 32784:20 := 96000000 // DRV Amplifier Settings / Velocity loop integral time
//         startup 32768:1 := 00 // FB Settings / Invert feedback direction
//       Term 16 (EL7211-9014) [EL7211-9014 1Ch. MDP742 Servo motor output stage with OCT (50V, 4.5A RMS) and STO input]
//         startup 32785:21 := 0E01 // DRV Motor Settings / Commutation offset
//         startup 32786:19 := 0000 // DRV Brake Settings / Emergency application timeout
//         startup 32784:51 := 0A00 // DRV Amplifier Settings / Stand still window
//         startup 32785:27 := D30C0000 // DRV Motor Settings / Motor speed limitation
//         startup 28688:11 := D007 // DRV Outputs / Torque limitation
//         startup 32784:19 := 4C01 // DRV Amplifier Settings / Current loop proportional gain
//         startup 32784:18 := 0500 // DRV Amplifier Settings / Current loop integral time
//         startup 32784:21 := 95000000 // DRV Amplifier Settings / Velocity loop proportional gain
//         startup 32784:20 := 96000000 // DRV Amplifier Settings / Velocity loop integral time
//         startup 32768:1 := 00 // FB Settings / Invert feedback direction
//       Term 17 (EL3022) [EL3022 2Ch. Ana. Input 4-20mA DIFF]
//       Term 18 (EL1809) [EL1809 16Ch. Dig. Input 24V, 3ms]
//       Term 19 (EL2904) [EL2904, 4 Ch. Safety Output 24V, 0.5A, TwinSAFE]
//         modules: Module 1 (FSOES), Module 2 (DO)
//       Term 20 (EL6631) [EL6631 PROFINET IO Controller]
//       Term 36 (EL9011) [EL9011 End Terminal]
//     Term 22 (EK1100) [EK1100 EtherCAT Coupler (2A E-Bus)]
//       Term 23 (EL7062) [EL7062-0000 2Ch. Stepper motor output stage (48V, 3A)]
//         startup 32785:27 := 8C000000 // DRV Motor Settings Ch.1 / Motor speed limitation
//         startup 32785:52 := E8030000 // DRV Motor Settings Ch.1 / Configured motor current
//         startup 32784:19 := 3200 // DRV Amplifier Settings Ch.1 / Current loop proportional gain
//         startup 32784:18 := 0900 // DRV Amplifier Settings Ch.1 / Current loop integral time
//         startup 32784:21 := 0B000000 // DRV Amplifier Settings Ch.1 / Velocity loop proportional gain
//         startup 32784:20 := 96000000 // DRV Amplifier Settings Ch.1 / Velocity loop integral time
//         startup 33041:27 := A0000000 // DRV Motor Settings Ch.2 / Motor speed limitation
//         startup 33041:52 := D0070000 // DRV Motor Settings Ch.2 / Configured motor current
//         startup 33040:19 := 2E00 // DRV Amplifier Settings Ch.2 / Current loop proportional gain
//         startup 33040:18 := 1400 // DRV Amplifier Settings Ch.2 / Current loop integral time
//         startup 33040:21 := 18000000 // DRV Amplifier Settings Ch.2 / Velocity loop proportional gain
//         startup 33040:20 := 96000000 // DRV Amplifier Settings Ch.2 / Velocity loop integral time
//       Term 24 (EL7062) [EL7062-0000 2Ch. Stepper motor output stage (48V, 3A)]
//         startup 32785:27 := 8C000000 // DRV Motor Settings Ch.1 / Motor speed limitation
//         startup 32785:52 := E8030000 // DRV Motor Settings Ch.1 / Configured motor current
//         startup 32784:19 := 3200 // DRV Amplifier Settings Ch.1 / Current loop proportional gain
//         startup 32784:18 := 0900 // DRV Amplifier Settings Ch.1 / Current loop integral time
//         startup 32784:21 := 0B000000 // DRV Amplifier Settings Ch.1 / Velocity loop proportional gain
//         startup 32784:20 := 96000000 // DRV Amplifier Settings Ch.1 / Velocity loop integral time
//         startup 33041:27 := A0000000 // DRV Motor Settings Ch.2 / Motor speed limitation
//         startup 33041:52 := D0070000 // DRV Motor Settings Ch.2 / Configured motor current
//         startup 33040:19 := 2E00 // DRV Amplifier Settings Ch.2 / Current loop proportional gain
//         startup 33040:18 := 1400 // DRV Amplifier Settings Ch.2 / Current loop integral time
//         startup 33040:21 := 18000000 // DRV Amplifier Settings Ch.2 / Velocity loop proportional gain
//         startup 33040:20 := 96000000 // DRV Amplifier Settings Ch.2 / Velocity loop integral time
//       Term 25 (EL7062) [EL7062-0000 2Ch. Stepper motor output stage (48V, 3A)]
//         startup 32785:27 := 8C000000 // DRV Motor Settings Ch.1 / Motor speed limitation
//         startup 32785:52 := E8030000 // DRV Motor Settings Ch.1 / Configured motor current
//         startup 32784:19 := 3200 // DRV Amplifier Settings Ch.1 / Current loop proportional gain
//         startup 32784:18 := 0900 // DRV Amplifier Settings Ch.1 / Current loop integral time
//         startup 32784:21 := 0B000000 // DRV Amplifier Settings Ch.1 / Velocity loop proportional gain
//         startup 32784:20 := 96000000 // DRV Amplifier Settings Ch.1 / Velocity loop integral time
//         startup 33041:27 := A0000000 // DRV Motor Settings Ch.2 / Motor speed limitation
//         startup 33041:52 := D0070000 // DRV Motor Settings Ch.2 / Configured motor current
//         startup 33040:19 := 2E00 // DRV Amplifier Settings Ch.2 / Current loop proportional gain
//         startup 33040:18 := 1400 // DRV Amplifier Settings Ch.2 / Current loop integral time
//         startup 33040:21 := 18000000 // DRV Amplifier Settings Ch.2 / Velocity loop proportional gain
//         startup 33040:20 := 96000000 // DRV Amplifier Settings Ch.2 / Velocity loop integral time
//       Term 26 (EL7062) [EL7062-0000 2Ch. Stepper motor output stage (48V, 3A)]
//         startup 32785:27 := 8C000000 // DRV Motor Settings Ch.1 / Motor speed limitation
//         startup 32785:52 := E8030000 // DRV Motor Settings Ch.1 / Configured motor current
//         startup 32784:19 := 3200 // DRV Amplifier Settings Ch.1 / Current loop proportional gain
//         startup 32784:18 := 0900 // DRV Amplifier Settings Ch.1 / Current loop integral time
//         startup 32784:21 := 0B000000 // DRV Amplifier Settings Ch.1 / Velocity loop proportional gain
//         startup 32784:20 := 96000000 // DRV Amplifier Settings Ch.1 / Velocity loop integral time
//         startup 33041:27 := A0000000 // DRV Motor Settings Ch.2 / Motor speed limitation
//         startup 33041:52 := D0070000 // DRV Motor Settings Ch.2 / Configured motor current
//         startup 33040:19 := 2E00 // DRV Amplifier Settings Ch.2 / Current loop proportional gain
//         startup 33040:18 := 1400 // DRV Amplifier Settings Ch.2 / Current loop integral time
//         startup 33040:21 := 18000000 // DRV Amplifier Settings Ch.2 / Velocity loop proportional gain
//         startup 33040:20 := 96000000 // DRV Amplifier Settings Ch.2 / Velocity loop integral time
//       Term 27 (EL7062) [EL7062-0000 2Ch. Stepper motor output stage (48V, 3A)]
//         startup 32785:27 := 8C000000 // DRV Motor Settings Ch.1 / Motor speed limitation
//         startup 32785:52 := E8030000 // DRV Motor Settings Ch.1 / Configured motor current
//         startup 32784:19 := 3200 // DRV Amplifier Settings Ch.1 / Current loop proportional gain
//         startup 32784:18 := 0900 // DRV Amplifier Settings Ch.1 / Current loop integral time
//         startup 32784:21 := 0B000000 // DRV Amplifier Settings Ch.1 / Velocity loop proportional gain
//         startup 32784:20 := 96000000 // DRV Amplifier Settings Ch.1 / Velocity loop integral time
//         startup 33041:27 := A0000000 // DRV Motor Settings Ch.2 / Motor speed limitation
//         startup 33041:52 := D0070000 // DRV Motor Settings Ch.2 / Configured motor current
//         startup 33040:19 := 2E00 // DRV Amplifier Settings Ch.2 / Current loop proportional gain
//         startup 33040:18 := 1400 // DRV Amplifier Settings Ch.2 / Current loop integral time
//         startup 33040:21 := 18000000 // DRV Amplifier Settings Ch.2 / Velocity loop proportional gain
//         startup 33040:20 := 96000000 // DRV Amplifier Settings Ch.2 / Velocity loop integral time
//       Term 28 (EL7062) [EL7062-0000 2Ch. Stepper motor output stage (48V, 3A)]
//         startup 32785:27 := 8C000000 // DRV Motor Settings Ch.1 / Motor speed limitation
//         startup 32785:52 := E8030000 // DRV Motor Settings Ch.1 / Configured motor current
//         startup 32784:19 := 3200 // DRV Amplifier Settings Ch.1 / Current loop proportional gain
//         startup 32784:18 := 0900 // DRV Amplifier Settings Ch.1 / Current loop integral time
//         startup 32784:21 := 0B000000 // DRV Amplifier Settings Ch.1 / Velocity loop proportional gain
//         startup 32784:20 := 96000000 // DRV Amplifier Settings Ch.1 / Velocity loop integral time
//         startup 33041:27 := A0000000 // DRV Motor Settings Ch.2 / Motor speed limitation
//         startup 33041:52 := D0070000 // DRV Motor Settings Ch.2 / Configured motor current
//         startup 33040:19 := 2E00 // DRV Amplifier Settings Ch.2 / Current loop proportional gain
//         startup 33040:18 := 1400 // DRV Amplifier Settings Ch.2 / Current loop integral time
//         startup 33040:21 := 18000000 // DRV Amplifier Settings Ch.2 / Velocity loop proportional gain
//         startup 33040:20 := 96000000 // DRV Amplifier Settings Ch.2 / Velocity loop integral time
//       Term 29 (EL7062) [EL7062-0000 2Ch. Stepper motor output stage (48V, 3A)]
//         startup 32785:27 := 8C000000 // DRV Motor Settings Ch.1 / Motor speed limitation
//         startup 32785:52 := E8030000 // DRV Motor Settings Ch.1 / Configured motor current
//         startup 32784:19 := 3200 // DRV Amplifier Settings Ch.1 / Current loop proportional gain
//         startup 32784:18 := 0900 // DRV Amplifier Settings Ch.1 / Current loop integral time
//         startup 32784:21 := 0B000000 // DRV Amplifier Settings Ch.1 / Velocity loop proportional gain
//         startup 32784:20 := 96000000 // DRV Amplifier Settings Ch.1 / Velocity loop integral time
//         startup 33041:27 := A0000000 // DRV Motor Settings Ch.2 / Motor speed limitation
//         startup 33041:52 := D0070000 // DRV Motor Settings Ch.2 / Configured motor current
//         startup 33040:19 := 2E00 // DRV Amplifier Settings Ch.2 / Current loop proportional gain
//         startup 33040:18 := 1400 // DRV Amplifier Settings Ch.2 / Current loop integral time
//         startup 33040:21 := 18000000 // DRV Amplifier Settings Ch.2 / Velocity loop proportional gain
//         startup 33040:20 := 96000000 // DRV Amplifier Settings Ch.2 / Velocity loop integral time
//       Term 30 (EL7062) [EL7062-0000 2Ch. Stepper motor output stage (48V, 3A)]
//         startup 32785:27 := 8C000000 // DRV Motor Settings Ch.1 / Motor speed limitation
//         startup 32785:52 := E8030000 // DRV Motor Settings Ch.1 / Configured motor current
//         startup 32784:19 := 3200 // DRV Amplifier Settings Ch.1 / Current loop proportional gain
//         startup 32784:18 := 0900 // DRV Amplifier Settings Ch.1 / Current loop integral time
//         startup 32784:21 := 0B000000 // DRV Amplifier Settings Ch.1 / Velocity loop proportional gain
//         startup 32784:20 := 96000000 // DRV Amplifier Settings Ch.1 / Velocity loop integral time
//         startup 33041:27 := A0000000 // DRV Motor Settings Ch.2 / Motor speed limitation
//         startup 33041:52 := D0070000 // DRV Motor Settings Ch.2 / Configured motor current
//         startup 33040:19 := 2E00 // DRV Amplifier Settings Ch.2 / Current loop proportional gain
//         startup 33040:18 := 1400 // DRV Amplifier Settings Ch.2 / Current loop integral time
//         startup 33040:21 := 18000000 // DRV Amplifier Settings Ch.2 / Velocity loop proportional gain
//         startup 33040:20 := 96000000 // DRV Amplifier Settings Ch.2 / Velocity loop integral time
//       Term 31 (EL7062) [EL7062-0000 2Ch. Stepper motor output stage (48V, 3A)]
//         startup 32785:27 := 8C000000 // DRV Motor Settings Ch.1 / Motor speed limitation
//         startup 32785:52 := E8030000 // DRV Motor Settings Ch.1 / Configured motor current
//         startup 32784:19 := 3200 // DRV Amplifier Settings Ch.1 / Current loop proportional gain
//         startup 32784:18 := 0900 // DRV Amplifier Settings Ch.1 / Current loop integral time
//         startup 32784:21 := 0B000000 // DRV Amplifier Settings Ch.1 / Velocity loop proportional gain
//         startup 32784:20 := 96000000 // DRV Amplifier Settings Ch.1 / Velocity loop integral time
//         startup 33041:27 := A0000000 // DRV Motor Settings Ch.2 / Motor speed limitation
//         startup 33041:52 := D0070000 // DRV Motor Settings Ch.2 / Configured motor current
//         startup 33040:19 := 2E00 // DRV Amplifier Settings Ch.2 / Current loop proportional gain
//         startup 33040:18 := 1400 // DRV Amplifier Settings Ch.2 / Current loop integral time
//         startup 33040:21 := 18000000 // DRV Amplifier Settings Ch.2 / Velocity loop proportional gain
//         startup 33040:20 := 96000000 // DRV Amplifier Settings Ch.2 / Velocity loop integral time
//       Term 32 (EL7062) [EL7062-0000 2Ch. Stepper motor output stage (48V, 3A)]
//         startup 32785:27 := 8C000000 // DRV Motor Settings Ch.1 / Motor speed limitation
//         startup 32785:52 := E8030000 // DRV Motor Settings Ch.1 / Configured motor current
//         startup 32784:19 := 3200 // DRV Amplifier Settings Ch.1 / Current loop proportional gain
//         startup 32784:18 := 0900 // DRV Amplifier Settings Ch.1 / Current loop integral time
//         startup 32784:21 := 0B000000 // DRV Amplifier Settings Ch.1 / Velocity loop proportional gain
//         startup 32784:20 := 96000000 // DRV Amplifier Settings Ch.1 / Velocity loop integral time
//         startup 33041:27 := A0000000 // DRV Motor Settings Ch.2 / Motor speed limitation
//         startup 33041:52 := D0070000 // DRV Motor Settings Ch.2 / Configured motor current
//         startup 33040:19 := 2E00 // DRV Amplifier Settings Ch.2 / Current loop proportional gain
//         startup 33040:18 := 1400 // DRV Amplifier Settings Ch.2 / Current loop integral time
//         startup 33040:21 := 18000000 // DRV Amplifier Settings Ch.2 / Velocity loop proportional gain
//         startup 33040:20 := 96000000 // DRV Amplifier Settings Ch.2 / Velocity loop integral time
//       Term 37 (EL9011) [EL9011 End Terminal]
//     Term 33 (AX8620-0000-0105) [AX8620-0000-0105]
//       Drive 34 (AX8108-0100-0106) [AX8108-0100-0106 (1Ch. 8A servo axis, STO)]
//         modules: Device, Device, Device, Device, Device, Device, Device, Device, Device, Device, Device (Safety), Device, Device, Device, Device, Device, Device, Device, Device, Device, Device, Device, Device, Device, Device, Device, Device, Device, Device, Device, Device, Ch A, Ch A, Ch A, Ch A, Ch A, Ch A, Ch A, Ch A, Ch A, Ch A, Ch A, Ch A, Ch A, Ch A, Ch A, Ch A, Ch A, Ch A, Ch A, Ch A, Ch A, Ch A, Ch A, Ch A, Ch A, Ch A, Ch A
//         startup 12992:1 := 414D383033322D78447831 // Ch A Motor parameters / Configured motor type
//         startup 24768:0 := FEFF // Ch A Interpolation sub mode select
//         startup 13000:5 := 0200 // Ch A Motor thermal model / Reaction
//         startup 13000:6 := 0000C841 // Ch A Motor thermal model / Partial fraction factor
//         startup 12992:12 := 00803B45 // Ch A Motor parameters / Motor rated speed
//         startup 12992:13 := 295C0F40 // Ch A Motor parameters / Motor rated torque
//         startup 24694:0 := 4C090000 // Ch A Motor standstill torque
//         startup 24800:0 := D007 // Ch A Positive torque/force limit value
//         startup 24801:0 := D007 // Ch A Negative torque/force limit value
//         startup 12288:6 := 4158383130382D303130302D30303030 // Ch A AxisMain parameters / Configured drive type
//         startup 12867:1 := 9A99D93F // Ch A TorqueCtrl parameters / Configured channel rated current
//         startup 12867:2 := 3333A340 // Ch A TorqueCtrl parameters / Configured channel peak current
//         startup 12867:7 := F4FD5440 // Ch A TorqueCtrl parameters / Iuvw max sum
//         startup 24672:0 := 08 // Ch A Modes of operation
//         startup 13023:0 := 0000 // Ch A Motor control mode
//         startup 12864:1 := 08F08043 // Ch A TorqueCtrl parameters mappable / Torque control proportional gain q
//         startup 12864:2 := 8A0E7C39 // Ch A TorqueCtrl parameters mappable / Torque control integral action time q
//         startup 12608:1 := ABCD313D // Ch A VeloCtrl parameters mappable / Velocity control proportional gain
//         startup 12608:2 := 6F12033C // Ch A VeloCtrl parameters mappable / Velocity control integral action time
//         startup 12608:3 := 00980546 // Ch A VeloCtrl parameters mappable / Bipolar velocity limit value
//         startup 12992:15 := 0100 // Ch A Motor parameters / Motor temperature sensor connection
//         startup 12611:4 := 0400 // Ch A VeloCtrl observer / Observer type
//         startup 24672:0 := 08 // Ch A Modes of operation
//         startup 12296:2 := 00 // Ch A AxisMain parameters encoder direction / Primary encoder direction
//     Box 1 (ifm IO-Link Master AL1333) [ifm IO-Link Master AL1333]
//       modules: Module 1 (IOL_In_4Byte), Module 2 (IOL_In_4Byte), Module 3 (IOL_In_4Byte), Module 4 (IOL_In_4Byte), Module 5 (IOL_In_4Byte), Module 6 (IOL_4/4_I/O-Bytes), Module 7 (IOL_4/4_I/O-Bytes), Module 8 (IOL_4/4_I/O-Bytes)
//   DEVICE Device 2 (EtherCAT Automation Protocol) (disabled), AmsNetId 192.168.0.162.3.1
//   DEVICE Device 5 (EL6631), AmsNetId 192.168.0.162.6.1
//     dl-pn1 [Keyence DL-PN1 PROFINET IO Device DL-PN1]
//       modules: Term 1 (DAP Module), Term 2 (DL-PN1), Term 3 (GT2-***)
// variable links:
//   Device 3 (EtherCAT) <-> Device 3 (EtherCAT)/Term 1 (EK1100)/Term 3 (EL6910)
//     Term 1 (EK1100)/Term 19 (EL2904)/Module 1 (FSOES)/RxPDO/FSOE <-> ConnectionInputs/TwinSafeGroup1.Term 31 (EL2904) - Module 1 (FSOES)_32 TxPDO
//     Term 1 (EK1100)/Term 19 (EL2904)/Module 1 (FSOES)/TxPDO/FSOE <-> ConnectionOutputs/TwinSafeGroup1.Term 31 (EL2904) - Module 1 (FSOES)_32 RxPDO
//     Term 1 (EK1100)/Term 7 (EL2904)/Module 1 (FSOES)/TxPDO/FSOE <-> ConnectionOutputs/TwinSafeGroup1.Term 19 (EL2904) - Module 1 (FSOES)_5 RxPDO
//     Term 1 (EK1100)/Term 8 (EL2904)/Module 1 (FSOES)/TxPDO/FSOE <-> ConnectionOutputs/TwinSafeGroup1.Term 20 (EL2904) - Module 1 (FSOES)_6 RxPDO
//     Term 1 (EK1100)/Term 4 (EL1918)/Module 1 (FSOE)/FSoE Inputs/FSOE <-> ConnectionOutputs/TwinSafeGroup1.Term 16 (EL1918) - Module 1 (FSOE)_1 RxPDO
//     Term 1 (EK1100)/Term 5 (EL1918)/Module 1 (FSOE)/FSoE Inputs/FSOE <-> ConnectionOutputs/TwinSafeGroup1.Term 17 (EL1918) - Module 1 (FSOE)_3 RxPDO
//     Term 33 (AX8620-0000-0105)/Drive 34 (AX8108-0100-0106)/Device (Safety)/FSoE Slave Connection 1 Master Message/ChA_Connection_Input.SAFEMOTION FSoE Connection_1 <-> ConnectionInputs/TwinSafeGroup1.Connection to Drive 46 (AX8108-0100-0106)_41 TxPDO
//     Term 33 (AX8620-0000-0105)/Drive 34 (AX8108-0100-0106)/Device (Safety)/FSoE Slave Connection 1 Slave Message/ChA_Connection_Input.SAFEMOTION FSoE Connection_1 <-> ConnectionOutputs/TwinSafeGroup1.Connection to Drive 46 (AX8108-0100-0106)_41 RxPDO
//   Device 3 (EtherCAT) <-> Device 3 (EtherCAT)/Term 1 (EK1100)/Term 4 (EL1918)
//     Term 1 (EK1100)/Term 3 (EL6910)/ConnectionInputs/TwinSafeGroup1.Term 16 (EL1918) - Module 1 (FSOE)_1 TxPDO <-> Module 1 (FSOE)/FSoE Outputs/FSOE
//   Device 3 (EtherCAT) <-> Device 3 (EtherCAT)/Term 1 (EK1100)/Term 5 (EL1918)
//     Term 1 (EK1100)/Term 3 (EL6910)/ConnectionInputs/TwinSafeGroup1.Term 17 (EL1918) - Module 1 (FSOE)_3 TxPDO <-> Module 1 (FSOE)/FSoE Outputs/FSOE
//   Device 3 (EtherCAT) <-> Device 3 (EtherCAT)/Term 1 (EK1100)/Term 6 (EL1918)
//     Term 1 (EK1100)/Term 3 (EL6910)/ConnectionInputs/TwinSafeGroup1.Term 18 (EL1918) - Module 1 (FSOE)_4 TxPDO <-> Module 1 (FSOE)/FSoE Outputs/FSOE
//     Term 1 (EK1100)/Term 3 (EL6910)/ConnectionOutputs/TwinSafeGroup1.Term 18 (EL1918) - Module 1 (FSOE)_4 RxPDO <-> Module 1 (FSOE)/FSoE Inputs/FSOE
//   Device 3 (EtherCAT) <-> Device 3 (EtherCAT)/Term 1 (EK1100)/Term 7 (EL2904)
//     Term 1 (EK1100)/Term 3 (EL6910)/ConnectionInputs/TwinSafeGroup1.Term 19 (EL2904) - Module 1 (FSOES)_5 TxPDO <-> Module 1 (FSOES)/RxPDO/FSOE
//   Device 3 (EtherCAT) <-> Device 3 (EtherCAT)/Term 1 (EK1100)/Term 8 (EL2904)
//     Term 1 (EK1100)/Term 3 (EL6910)/ConnectionInputs/TwinSafeGroup1.Term 20 (EL2904) - Module 1 (FSOES)_6 TxPDO <-> Module 1 (FSOES)/RxPDO/FSOE
//   Device 3 (EtherCAT) <-> Device 3 (EtherCAT)/Term 33 (AX8620-0000-0105)
//     Term 33 (AX8620-0000-0105)/Drive 34 (AX8108-0100-0106)/Device/DeviceMain Outputs/Power supply controlword <-> PSM Controlword for axis/Controlword for axis
//   Device 3 (EtherCAT) <-> Device 6 (EtherCAT)/Box 10 (AMI8000-0100)
//     Term 1 (EK1100)/Term 3 (EL6910)/ConnectionOutputs/TwinSafeGroup1.Connection to Box 10 (AMI8000-0100)_111 RxPDO <-> Module 1 (SAFETY)/SAFETY FSoE Connection 1 Send Message/Message_1
//   Device 3 (EtherCAT) <-> Device 6 (EtherCAT)/Box 11 (AMI8000-0100)
//     Term 1 (EK1100)/Term 3 (EL6910)/ConnectionOutputs/TwinSafeGroup1.Connection to Box 11 (AMI8000-0100)_106 RxPDO <-> Module 1 (SAFETY)/SAFETY FSoE Connection 1 Send Message/Message_1
//   Device 3 (EtherCAT) <-> Device 6 (EtherCAT)/Box 12 (AMI8000-0100)
//     Term 1 (EK1100)/Term 3 (EL6910)/ConnectionInputs/TwinSafeGroup1.Connection to Box 12 (AMI8000-0100)_105 TxPDO <-> Module 1 (SAFETY)/SAFETY FSoE Connection 1 Receive Message/Message_1
//   Device 3 (EtherCAT) <-> Device 6 (EtherCAT)/Box 9 (AMI8000-0100)
//     Term 1 (EK1100)/Term 3 (EL6910)/ConnectionInputs/TwinSafeGroup1.Connection to Box 9 (AMI8000-0100)_102 TxPDO <-> Module 1 (SAFETY)/SAFETY FSoE Connection 1 Receive Message/Message_1
//     Term 1 (EK1100)/Term 3 (EL6910)/ConnectionOutputs/TwinSafeGroup1.Connection to Box 9 (AMI8000-0100)_102 RxPDO <-> Module 1 (SAFETY)/SAFETY FSoE Connection 1 Send Message/Message_1
//   Device 6 (EtherCAT) <-> Device 3 (EtherCAT)/Term 1 (EK1100)/Term 3 (EL6910)
//     Box 10 (AMI8000-0100)/Module 1 (SAFETY)/SAFETY FSoE Connection 1 Receive Message/Message_1 <-> ConnectionInputs/TwinSafeGroup1.Connection to Box 10 (AMI8000-0100)_111 TxPDO
//     Box 11 (AMI8000-0100)/Module 1 (SAFETY)/SAFETY FSoE Connection 1 Receive Message/Message_1 <-> ConnectionInputs/TwinSafeGroup1.Connection to Box 11 (AMI8000-0100)_106 TxPDO
//     Box 8 (AMI8000-0100)/Module 1 (SAFETY)/SAFETY FSoE Connection 1 Receive Message/Message_1 <-> ConnectionInputs/TwinSafeGroup1.Connection to Box 8 (AMI8000-0100)_101 TxPDO
//     Box 12 (AMI8000-0100)/Module 1 (SAFETY)/SAFETY FSoE Connection 1 Send Message/Message_1 <-> ConnectionOutputs/TwinSafeGroup1.Connection to Box 12 (AMI8000-0100)_105 RxPDO
//     Box 8 (AMI8000-0100)/Module 1 (SAFETY)/SAFETY FSoE Connection 1 Send Message/Message_1 <-> ConnectionOutputs/TwinSafeGroup1.Connection to Box 8 (AMI8000-0100)_101 RxPDO
//   NC-Task 1 SAF/Axes/M1 Motor - SR Vertical <-> Device 3 (EtherCAT)/Term 33 (AX8620-0000-0105)/Drive 34 (AX8108-0100-0106)
//     Drive/Inputs/In/nDataIn1 <-> Ch A/Ch A PositionControl Inputs/Ch A Following error actual value
//     Drive/Inputs/In/nDataIn3[0] <-> Ch A/Ch A TorqueControl Inputs/Ch A Torque/force actual value
//     Drive/Inputs/In/nDcOutputTime <-> InfoData/DcOutputShift
//     Drive/Inputs/In/nState1 <-> Ch A/Ch A AxisMain Inputs/Ch A Statusword
//     Drive/Inputs/In/nState2 <-> Ch A/Ch A AxisMain Inputs/Ch A Statusword @bit 8
//     Drive/Inputs/In/nState4 @bit 1 <-> WcState/InputToggle0
//     Drive/Inputs/In/nState4 <-> WcState/WcState0
//     Drive/Outputs/Out/nCtrl1 <-> Ch A/Ch A AxisMain Outputs/Ch A Controlword
//     Drive/Outputs/Out/nCtrl2 <-> Ch A/Ch A AxisMain Outputs/Ch A Controlword @bit 8
//     Drive/Outputs/Out/nDataOut1 <-> Ch A/Ch A Interpolator Outputs/Ch A Target position
//     Drive/Outputs/Out/nDataOut2 <-> Ch A/Ch A Interpolator Outputs/Ch A Target velocity
//     Enc/Inputs/In/nDataIn1 <-> Ch A/Ch A AxisMain Inputs/Ch A Position actual value
//     Enc/Inputs/In/nDataIn7 <-> Ch A/Ch A AxisMain Inputs/Ch A Velocity actual value
//     Enc/Inputs/In/nDcInputTime <-> InfoData/DcInputShift
//     Enc/Inputs/In/nState2 @bit 5 <-> Ch A/Ch A AxisMain Inputs/Position actual value invalid
//     Enc/Inputs/In/nState4 @bit 1 <-> WcState/InputToggle0
//     Enc/Inputs/In/nState4 <-> WcState/WcState0
//   NC-Task 1 SAF/Axes/M2 Motor - SC Vertical <-> Device 3 (EtherCAT)/Term 1 (EK1100)/Term 15 (EL7211-9014)
//     Drive/Inputs/In/nDataIn1 <-> DRV Following error actual value/Following error actual value
//     Drive/Inputs/In/nDataIn3[0] <-> DRV Torque actual value/Torque actual value
//     Drive/Inputs/In/nDcOutputTime <-> InfoData/DcOutputShift
//     Drive/Inputs/In/nState1 <-> DRV Statusword/Statusword
//     Drive/Inputs/In/nState2 <-> DRV Statusword/Statusword @bit 8
//     Drive/Inputs/In/nState4 @bit 1 <-> WcState/InputToggle
//     Drive/Inputs/In/nState4 <-> WcState/WcState
//     Drive/Outputs/Out/nCtrl1 <-> DRV Controlword/Controlword
//     Drive/Outputs/Out/nCtrl2 <-> DRV Controlword/Controlword @bit 8
//     Drive/Outputs/Out/nDataOut1 <-> DRV Target position/Target position
//     Drive/Outputs/Out/nDataOut2 <-> DRV Target velocity/Target velocity
//     Drive/Outputs/Out/nDataOut4 <-> DRV Target torque/Target torque
//     Enc/Inputs/In/nDataIn1 <-> FB Position/Position
//     Enc/Inputs/In/nDcInputTime <-> InfoData/DcInputShift
//     Enc/Inputs/In/nState4 @bit 1 <-> WcState/InputToggle
//     Enc/Inputs/In/nState4 <-> WcState/WcState
//   NC-Task 1 SAF/Axes/M3 Motor - SC Horizontal <-> Device 3 (EtherCAT)/Term 1 (EK1100)/Term 16 (EL7211-9014)
//     Drive/Inputs/In/nDataIn1 <-> DRV Following error actual value/Following error actual value
//     Drive/Inputs/In/nDataIn3[0] <-> DRV Torque actual value/Torque actual value
//     Drive/Inputs/In/nDcOutputTime <-> InfoData/DcOutputShift
//     Drive/Inputs/In/nState1 <-> DRV Statusword/Statusword
//     Drive/Inputs/In/nState2 <-> DRV Statusword/Statusword @bit 8
//     Drive/Inputs/In/nState4 @bit 1 <-> WcState/InputToggle
//     Drive/Inputs/In/nState4 <-> WcState/WcState
//     Drive/Outputs/Out/nCtrl1 <-> DRV Controlword/Controlword
//     Drive/Outputs/Out/nCtrl2 <-> DRV Controlword/Controlword @bit 8
//     Drive/Outputs/Out/nDataOut1 <-> DRV Target position/Target position
//     Drive/Outputs/Out/nDataOut2 <-> DRV Target velocity/Target velocity
//     Drive/Outputs/Out/nDataOut4 <-> DRV Target torque/Target torque
//     Enc/Inputs/In/nDataIn1 <-> FB Position/Position
//     Enc/Inputs/In/nDcInputTime <-> InfoData/DcInputShift
//     Enc/Inputs/In/nState4 @bit 1 <-> WcState/InputToggle
//     Enc/Inputs/In/nState4 <-> WcState/WcState
//   NC-Task 1 SAF/Axes/M4 Motor - Valve 1 <-> Device 6 (EtherCAT)/Box 8 (AMI8000-0100)
//     Drive/Inputs/In/nDataIn1 <-> DRV Following error actual value/Following error actual value
//     Drive/Inputs/In/nDcOutputTime <-> InfoData/DcOutputShift
//     Drive/Inputs/In/nState1 <-> DRV Statusword/Statusword
//     Drive/Inputs/In/nState2 <-> DRV Statusword/Statusword @bit 8
//     Drive/Inputs/In/nState4 @bit 1 <-> WcState/InputToggle
//     Drive/Inputs/In/nState4 <-> WcState/WcState
//     Drive/Outputs/Out/nCtrl1 <-> DRV Controlword/Controlword
//     Drive/Outputs/Out/nCtrl2 <-> DRV Controlword/Controlword @bit 8
//     Drive/Outputs/Out/nDataOut1 <-> DRV Target position/Target position
//     Enc/Inputs/In/nDataIn1 <-> FB Position/Position
//     Enc/Inputs/In/nDcInputTime <-> InfoData/DcInputShift
//     Enc/Inputs/In/nState4 @bit 1 <-> WcState/InputToggle
//     Enc/Inputs/In/nState4 <-> WcState/WcState
//   NC-Task 1 SAF/Axes/M5 Motor - Valve 2 <-> Device 6 (EtherCAT)/Box 9 (AMI8000-0100)
//     Drive/Inputs/In/nDataIn1 <-> DRV Following error actual value/Following error actual value
//     Drive/Inputs/In/nDcOutputTime <-> InfoData/DcOutputShift
//     Drive/Inputs/In/nState1 <-> DRV Statusword/Statusword
//     Drive/Inputs/In/nState2 <-> DRV Statusword/Statusword @bit 8
//     Drive/Inputs/In/nState4 @bit 1 <-> WcState/InputToggle
//     Drive/Inputs/In/nState4 <-> WcState/WcState
//     Drive/Outputs/Out/nCtrl1 <-> DRV Controlword/Controlword
//     Drive/Outputs/Out/nCtrl2 <-> DRV Controlword/Controlword @bit 8
//     Drive/Outputs/Out/nDataOut1 <-> DRV Target position/Target position
//     Enc/Inputs/In/nDataIn1 <-> FB Position/Position
//     Enc/Inputs/In/nDcInputTime <-> InfoData/DcInputShift
//     Enc/Inputs/In/nState4 @bit 1 <-> WcState/InputToggle
//     Enc/Inputs/In/nState4 <-> WcState/WcState
//   NC-Task 1 SAF/Axes/M6 Motor - Valve 3 <-> Device 6 (EtherCAT)/Box 10 (AMI8000-0100)
//     Drive/Inputs/In/nDataIn1 <-> DRV Following error actual value/Following error actual value
//     Drive/Inputs/In/nDcOutputTime <-> InfoData/DcOutputShift
//     Drive/Inputs/In/nState1 <-> DRV Statusword/Statusword
//     Drive/Inputs/In/nState2 <-> DRV Statusword/Statusword @bit 8
//     Drive/Inputs/In/nState4 @bit 1 <-> WcState/InputToggle
//     Drive/Inputs/In/nState4 <-> WcState/WcState
//     Drive/Outputs/Out/nCtrl1 <-> DRV Controlword/Controlword
//     Drive/Outputs/Out/nCtrl2 <-> DRV Controlword/Controlword @bit 8
//     Drive/Outputs/Out/nDataOut1 <-> DRV Target position/Target position
//     Enc/Inputs/In/nDataIn1 <-> FB Position/Position
//     Enc/Inputs/In/nDcInputTime <-> InfoData/DcInputShift
//     Enc/Inputs/In/nState4 @bit 1 <-> WcState/InputToggle
//     Enc/Inputs/In/nState4 <-> WcState/WcState
//   NC-Task 1 SAF/Axes/M7 Motor - Valve 4 <-> Device 6 (EtherCAT)/Box 11 (AMI8000-0100)
//     Drive/Inputs/In/nDataIn1 <-> DRV Following error actual value/Following error actual value
//     Drive/Inputs/In/nDcOutputTime <-> InfoData/DcOutputShift
//     Drive/Inputs/In/nState1 <-> DRV Statusword/Statusword
//     Drive/Inputs/In/nState2 <-> DRV Statusword/Statusword @bit 8
//     Drive/Inputs/In/nState4 @bit 1 <-> WcState/InputToggle
//     Drive/Inputs/In/nState4 <-> WcState/WcState
//     Drive/Outputs/Out/nCtrl1 <-> DRV Controlword/Controlword
//     Drive/Outputs/Out/nCtrl2 <-> DRV Controlword/Controlword @bit 8
//     Drive/Outputs/Out/nDataOut1 <-> DRV Target position/Target position
//     Enc/Inputs/In/nDataIn1 <-> FB Position/Position
//     Enc/Inputs/In/nDcInputTime <-> InfoData/DcInputShift
//     Enc/Inputs/In/nState4 @bit 1 <-> WcState/InputToggle
//     Enc/Inputs/In/nState4 <-> WcState/WcState
//   NC-Task 1 SAF/Axes/M8 Motor - Valve 5 <-> Device 6 (EtherCAT)/Box 12 (AMI8000-0100)
//     Drive/Inputs/In/nDataIn1 <-> DRV Following error actual value/Following error actual value
//     Drive/Inputs/In/nDcOutputTime <-> InfoData/DcOutputShift
//     Drive/Inputs/In/nState1 <-> DRV Statusword/Statusword
//     Drive/Inputs/In/nState2 <-> DRV Statusword/Statusword @bit 8
//     Drive/Inputs/In/nState4 @bit 1 <-> WcState/InputToggle
//     Drive/Inputs/In/nState4 <-> WcState/WcState
//     Drive/Outputs/Out/nCtrl1 <-> DRV Controlword/Controlword
//     Drive/Outputs/Out/nCtrl2 <-> DRV Controlword/Controlword @bit 8
//     Drive/Outputs/Out/nDataOut1 <-> DRV Target position/Target position
//     Enc/Inputs/In/nDataIn1 <-> FB Position/Position
//     Enc/Inputs/In/nDcInputTime <-> InfoData/DcInputShift
//     Enc/Inputs/In/nState4 @bit 1 <-> WcState/InputToggle
//     Enc/Inputs/In/nState4 <-> WcState/WcState
//   NC-Task 1 SAF/Axes/Pump 1 - Linear <-> Device 3 (EtherCAT)/Term 22 (EK1100)/Term 23 (EL7062)
//     Drive/Inputs/In/nDataIn1 <-> DRV Following error actual value Channel 1/Following error actual value
//     Drive/Inputs/In/nDcOutputTime <-> InfoData/DcOutputShift
//     Drive/Inputs/In/nState1 <-> DRV Statusword Channel 1/Statusword
//     Drive/Inputs/In/nState2 <-> DRV Statusword Channel 1/Statusword @bit 8
//     Drive/Inputs/In/nState4 @bit 1 <-> WcState/InputToggle
//     Drive/Inputs/In/nState4 <-> WcState/WcState
//     Drive/Outputs/Out/nCtrl1 <-> DRV Controlword Channel 1/Controlword
//     Drive/Outputs/Out/nCtrl2 <-> DRV Controlword Channel 1/Controlword @bit 8
//     Drive/Outputs/Out/nDataOut1 <-> DRV Target position Channel 1/Target position
//     Enc/Inputs/In/nDataIn1 <-> FB Position Channel 1/Position
//     Enc/Inputs/In/nDcInputTime <-> InfoData/DcInputShift
//     Enc/Inputs/In/nState4 @bit 1 <-> WcState/InputToggle
//     Enc/Inputs/In/nState4 <-> WcState/WcState
//   NC-Task 1 SAF/Axes/Pump 1 - Rotary <-> Device 3 (EtherCAT)/Term 22 (EK1100)/Term 23 (EL7062)
//     Drive/Inputs/In/nDataIn1 <-> DRV Following error actual value Channel 2/Following error actual value
//     Drive/Inputs/In/nDcOutputTime <-> InfoData/DcOutputShift
//     Drive/Inputs/In/nState1 <-> DRV Statusword Channel 2/Statusword
//     Drive/Inputs/In/nState2 <-> DRV Statusword Channel 2/Statusword @bit 8
//     Drive/Inputs/In/nState4 @bit 1 <-> WcState/InputToggle
//     Drive/Inputs/In/nState4 <-> WcState/WcState
//     Drive/Outputs/Out/nCtrl1 <-> DRV Controlword Channel 2/Controlword
//     Drive/Outputs/Out/nCtrl2 <-> DRV Controlword Channel 2/Controlword @bit 8
//     Drive/Outputs/Out/nDataOut1 <-> DRV Target position Channel 2/Target position
//     Enc/Inputs/In/nDataIn1 <-> FB Position Channel 2/Position
//     Enc/Inputs/In/nDcInputTime <-> InfoData/DcInputShift
//     Enc/Inputs/In/nState4 @bit 1 <-> WcState/InputToggle
//     Enc/Inputs/In/nState4 <-> WcState/WcState
//   NC-Task 1 SAF/Axes/Pump 10 - Linear <-> Device 3 (EtherCAT)/Term 22 (EK1100)/Term 32 (EL7062)
//     Drive/Inputs/In/nDataIn1 <-> DRV Following error actual value Channel 1/Following error actual value
//     Drive/Inputs/In/nDcOutputTime <-> InfoData/DcOutputShift
//     Drive/Inputs/In/nState1 <-> DRV Statusword Channel 1/Statusword
//     Drive/Inputs/In/nState2 <-> DRV Statusword Channel 1/Statusword @bit 8
//     Drive/Inputs/In/nState4 @bit 1 <-> WcState/InputToggle
//     Drive/Inputs/In/nState4 <-> WcState/WcState
//     Drive/Outputs/Out/nCtrl1 <-> DRV Controlword Channel 1/Controlword
//     Drive/Outputs/Out/nCtrl2 <-> DRV Controlword Channel 1/Controlword @bit 8
//     Drive/Outputs/Out/nDataOut1 <-> DRV Target position Channel 1/Target position
//     Enc/Inputs/In/nDataIn1 <-> FB Position Channel 1/Position
//     Enc/Inputs/In/nDcInputTime <-> InfoData/DcInputShift
//     Enc/Inputs/In/nState4 @bit 1 <-> WcState/InputToggle
//     Enc/Inputs/In/nState4 <-> WcState/WcState
//   NC-Task 1 SAF/Axes/Pump 10 - Rotary <-> Device 3 (EtherCAT)/Term 22 (EK1100)/Term 32 (EL7062)
//     Drive/Inputs/In/nDataIn1 <-> DRV Following error actual value Channel 2/Following error actual value
//     Drive/Inputs/In/nDcOutputTime <-> InfoData/DcOutputShift
//     Drive/Inputs/In/nState1 <-> DRV Statusword Channel 2/Statusword
//     Drive/Inputs/In/nState2 <-> DRV Statusword Channel 2/Statusword @bit 8
//     Drive/Inputs/In/nState4 @bit 1 <-> WcState/InputToggle
//     Drive/Inputs/In/nState4 <-> WcState/WcState
//     Drive/Outputs/Out/nCtrl1 <-> DRV Controlword Channel 2/Controlword
//     Drive/Outputs/Out/nCtrl2 <-> DRV Controlword Channel 2/Controlword @bit 8
//     Drive/Outputs/Out/nDataOut1 <-> DRV Target position Channel 2/Target position
//     Enc/Inputs/In/nDataIn1 <-> FB Position Channel 2/Position
//     Enc/Inputs/In/nDcInputTime <-> InfoData/DcInputShift
//     Enc/Inputs/In/nState4 @bit 1 <-> WcState/InputToggle
//     Enc/Inputs/In/nState4 <-> WcState/WcState
//   NC-Task 1 SAF/Axes/Pump 2 - Linear <-> Device 3 (EtherCAT)/Term 22 (EK1100)/Term 24 (EL7062)
//     Drive/Inputs/In/nDataIn1 <-> DRV Following error actual value Channel 1/Following error actual value
//     Drive/Inputs/In/nDcOutputTime <-> InfoData/DcOutputShift
//     Drive/Inputs/In/nState1 <-> DRV Statusword Channel 1/Statusword
//     Drive/Inputs/In/nState2 <-> DRV Statusword Channel 1/Statusword @bit 8
//     Drive/Inputs/In/nState4 @bit 1 <-> WcState/InputToggle
//     Drive/Inputs/In/nState4 <-> WcState/WcState
//     Drive/Outputs/Out/nCtrl1 <-> DRV Controlword Channel 1/Controlword
//     Drive/Outputs/Out/nCtrl2 <-> DRV Controlword Channel 1/Controlword @bit 8
//     Drive/Outputs/Out/nDataOut1 <-> DRV Target position Channel 1/Target position
//     Enc/Inputs/In/nDataIn1 <-> FB Position Channel 1/Position
//     Enc/Inputs/In/nDcInputTime <-> InfoData/DcInputShift
//     Enc/Inputs/In/nState4 @bit 1 <-> WcState/InputToggle
//     Enc/Inputs/In/nState4 <-> WcState/WcState
//   NC-Task 1 SAF/Axes/Pump 2 - Rotary <-> Device 3 (EtherCAT)/Term 22 (EK1100)/Term 24 (EL7062)
//     Drive/Inputs/In/nDataIn1 <-> DRV Following error actual value Channel 2/Following error actual value
//     Drive/Inputs/In/nDcOutputTime <-> InfoData/DcOutputShift
//     Drive/Inputs/In/nState1 <-> DRV Statusword Channel 2/Statusword
//     Drive/Inputs/In/nState2 <-> DRV Statusword Channel 2/Statusword @bit 8
//     Drive/Inputs/In/nState4 @bit 1 <-> WcState/InputToggle
//     Drive/Inputs/In/nState4 <-> WcState/WcState
//     Drive/Outputs/Out/nCtrl1 <-> DRV Controlword Channel 2/Controlword
//     Drive/Outputs/Out/nCtrl2 <-> DRV Controlword Channel 2/Controlword @bit 8
//     Drive/Outputs/Out/nDataOut1 <-> DRV Target position Channel 2/Target position
//     Enc/Inputs/In/nDataIn1 <-> FB Position Channel 2/Position
//     Enc/Inputs/In/nDcInputTime <-> InfoData/DcInputShift
//     Enc/Inputs/In/nState4 @bit 1 <-> WcState/InputToggle
//     Enc/Inputs/In/nState4 <-> WcState/WcState
//   NC-Task 1 SAF/Axes/Pump 3 - Linear <-> Device 3 (EtherCAT)/Term 22 (EK1100)/Term 25 (EL7062)
//     Drive/Inputs/In/nDataIn1 <-> DRV Following error actual value Channel 1/Following error actual value
//     Drive/Inputs/In/nDcOutputTime <-> InfoData/DcOutputShift
//     Drive/Inputs/In/nState1 <-> DRV Statusword Channel 1/Statusword
//     Drive/Inputs/In/nState2 <-> DRV Statusword Channel 1/Statusword @bit 8
//     Drive/Inputs/In/nState4 @bit 1 <-> WcState/InputToggle
//     Drive/Inputs/In/nState4 <-> WcState/WcState
//     Drive/Outputs/Out/nCtrl1 <-> DRV Controlword Channel 1/Controlword
//     Drive/Outputs/Out/nCtrl2 <-> DRV Controlword Channel 1/Controlword @bit 8
//     Drive/Outputs/Out/nDataOut1 <-> DRV Target position Channel 1/Target position
//     Enc/Inputs/In/nDataIn1 <-> FB Position Channel 1/Position
//     Enc/Inputs/In/nDcInputTime <-> InfoData/DcInputShift
//     Enc/Inputs/In/nState4 @bit 1 <-> WcState/InputToggle
//     Enc/Inputs/In/nState4 <-> WcState/WcState
//   NC-Task 1 SAF/Axes/Pump 3 - Rotary <-> Device 3 (EtherCAT)/Term 22 (EK1100)/Term 25 (EL7062)
//     Drive/Inputs/In/nDataIn1 <-> DRV Following error actual value Channel 2/Following error actual value
//     Drive/Inputs/In/nDcOutputTime <-> InfoData/DcOutputShift
//     Drive/Inputs/In/nState1 <-> DRV Statusword Channel 2/Statusword
//     Drive/Inputs/In/nState2 <-> DRV Statusword Channel 2/Statusword @bit 8
//     Drive/Inputs/In/nState4 @bit 1 <-> WcState/InputToggle
//     Drive/Inputs/In/nState4 <-> WcState/WcState
//     Drive/Outputs/Out/nCtrl1 <-> DRV Controlword Channel 2/Controlword
//     Drive/Outputs/Out/nCtrl2 <-> DRV Controlword Channel 2/Controlword @bit 8
//     Drive/Outputs/Out/nDataOut1 <-> DRV Target position Channel 2/Target position
//     Drive/Outputs/Out/nDataOut2 <-> DRV Target velocity Channel 2/Target velocity
//     Enc/Inputs/In/nDataIn1 <-> FB Position Channel 2/Position
//     Enc/Inputs/In/nDcInputTime <-> InfoData/DcInputShift
//     Enc/Inputs/In/nState4 @bit 1 <-> WcState/InputToggle
//     Enc/Inputs/In/nState4 <-> WcState/WcState
//   NC-Task 1 SAF/Axes/Pump 4 - Linear <-> Device 3 (EtherCAT)/Term 22 (EK1100)/Term 26 (EL7062)
//     Drive/Inputs/In/nDataIn1 <-> DRV Following error actual value Channel 1/Following error actual value
//     Drive/Inputs/In/nDcOutputTime <-> InfoData/DcOutputShift
//     Drive/Inputs/In/nState1 <-> DRV Statusword Channel 1/Statusword
//     Drive/Inputs/In/nState2 <-> DRV Statusword Channel 1/Statusword @bit 8
//     Drive/Inputs/In/nState4 @bit 1 <-> WcState/InputToggle
//     Drive/Inputs/In/nState4 <-> WcState/WcState
//     Drive/Outputs/Out/nCtrl1 <-> DRV Controlword Channel 1/Controlword
//     Drive/Outputs/Out/nCtrl2 <-> DRV Controlword Channel 1/Controlword @bit 8
//     Drive/Outputs/Out/nDataOut1 <-> DRV Target position Channel 1/Target position
//     Enc/Inputs/In/nDataIn1 <-> FB Position Channel 1/Position
//     Enc/Inputs/In/nDcInputTime <-> InfoData/DcInputShift
//     Enc/Inputs/In/nState4 @bit 1 <-> WcState/InputToggle
//     Enc/Inputs/In/nState4 <-> WcState/WcState
//   NC-Task 1 SAF/Axes/Pump 4 - Rotary <-> Device 3 (EtherCAT)/Term 22 (EK1100)/Term 26 (EL7062)
//     Drive/Inputs/In/nDataIn1 <-> DRV Following error actual value Channel 2/Following error actual value
//     Drive/Inputs/In/nDcOutputTime <-> InfoData/DcOutputShift
//     Drive/Inputs/In/nState1 <-> DRV Statusword Channel 2/Statusword
//     Drive/Inputs/In/nState2 <-> DRV Statusword Channel 2/Statusword @bit 8
//     Drive/Inputs/In/nState4 @bit 1 <-> WcState/InputToggle
//     Drive/Inputs/In/nState4 <-> WcState/WcState
//     Drive/Outputs/Out/nCtrl1 <-> DRV Controlword Channel 2/Controlword
//     Drive/Outputs/Out/nCtrl2 <-> DRV Controlword Channel 2/Controlword @bit 8
//     Drive/Outputs/Out/nDataOut1 <-> DRV Target position Channel 2/Target position
//     Enc/Inputs/In/nDataIn1 <-> FB Position Channel 2/Position
//     Enc/Inputs/In/nDcInputTime <-> InfoData/DcInputShift
//     Enc/Inputs/In/nState4 @bit 1 <-> WcState/InputToggle
//     Enc/Inputs/In/nState4 <-> WcState/WcState
//   NC-Task 1 SAF/Axes/Pump 5 - Linear <-> Device 3 (EtherCAT)/Term 22 (EK1100)/Term 27 (EL7062)
//     Drive/Inputs/In/nDataIn1 <-> DRV Following error actual value Channel 1/Following error actual value
//     Drive/Inputs/In/nDcOutputTime <-> InfoData/DcOutputShift
//     Drive/Inputs/In/nState1 <-> DRV Statusword Channel 1/Statusword
//     Drive/Inputs/In/nState2 <-> DRV Statusword Channel 1/Statusword @bit 8
//     Drive/Inputs/In/nState4 @bit 1 <-> WcState/InputToggle
//     Drive/Inputs/In/nState4 <-> WcState/WcState
//     Drive/Outputs/Out/nCtrl1 <-> DRV Controlword Channel 1/Controlword
//     Drive/Outputs/Out/nCtrl2 <-> DRV Controlword Channel 1/Controlword @bit 8
//     Drive/Outputs/Out/nDataOut1 <-> DRV Target position Channel 1/Target position
//     Enc/Inputs/In/nDataIn1 <-> FB Position Channel 1/Position
//     Enc/Inputs/In/nDcInputTime <-> InfoData/DcInputShift
//     Enc/Inputs/In/nState4 @bit 1 <-> WcState/InputToggle
//     Enc/Inputs/In/nState4 <-> WcState/WcState
//   NC-Task 1 SAF/Axes/Pump 5 - Rotary <-> Device 3 (EtherCAT)/Term 22 (EK1100)/Term 27 (EL7062)
//     Drive/Inputs/In/nDataIn1 <-> DRV Following error actual value Channel 2/Following error actual value
//     Drive/Inputs/In/nDcOutputTime <-> InfoData/DcOutputShift
//     Drive/Inputs/In/nState1 <-> DRV Statusword Channel 2/Statusword
//     Drive/Inputs/In/nState2 <-> DRV Statusword Channel 2/Statusword @bit 8
//     Drive/Inputs/In/nState4 @bit 1 <-> WcState/InputToggle
//     Drive/Inputs/In/nState4 <-> WcState/WcState
//     Drive/Outputs/Out/nCtrl1 <-> DRV Controlword Channel 2/Controlword
//     Drive/Outputs/Out/nCtrl2 <-> DRV Controlword Channel 2/Controlword @bit 8
//     Drive/Outputs/Out/nDataOut1 <-> DRV Target position Channel 2/Target position
//     Enc/Inputs/In/nDataIn1 <-> FB Position Channel 2/Position
//     Enc/Inputs/In/nDcInputTime <-> InfoData/DcInputShift
//     Enc/Inputs/In/nState4 @bit 1 <-> WcState/InputToggle
//     Enc/Inputs/In/nState4 <-> WcState/WcState
//   NC-Task 1 SAF/Axes/Pump 6 - Linear <-> Device 3 (EtherCAT)/Term 22 (EK1100)/Term 28 (EL7062)
//     Drive/Inputs/In/nDataIn1 <-> DRV Following error actual value Channel 1/Following error actual value
//     Drive/Inputs/In/nDcOutputTime <-> InfoData/DcOutputShift
//     Drive/Inputs/In/nState1 <-> DRV Statusword Channel 1/Statusword
//     Drive/Inputs/In/nState2 <-> DRV Statusword Channel 1/Statusword @bit 8
//     Drive/Inputs/In/nState4 @bit 1 <-> WcState/InputToggle
//     Drive/Inputs/In/nState4 <-> WcState/WcState
//     Drive/Outputs/Out/nCtrl1 <-> DRV Controlword Channel 1/Controlword
//     Drive/Outputs/Out/nCtrl2 <-> DRV Controlword Channel 1/Controlword @bit 8
//     Drive/Outputs/Out/nDataOut1 <-> DRV Target position Channel 1/Target position
//     Enc/Inputs/In/nDataIn1 <-> FB Position Channel 1/Position
//     Enc/Inputs/In/nDcInputTime <-> InfoData/DcInputShift
//     Enc/Inputs/In/nState4 @bit 1 <-> WcState/InputToggle
//     Enc/Inputs/In/nState4 <-> WcState/WcState
//   NC-Task 1 SAF/Axes/Pump 6 - Rotary <-> Device 3 (EtherCAT)/Term 22 (EK1100)/Term 28 (EL7062)
//     Drive/Inputs/In/nDataIn1 <-> DRV Following error actual value Channel 2/Following error actual value
//     Drive/Inputs/In/nDcOutputTime <-> InfoData/DcOutputShift
//     Drive/Inputs/In/nState1 <-> DRV Statusword Channel 2/Statusword
//     Drive/Inputs/In/nState2 <-> DRV Statusword Channel 2/Statusword @bit 8
//     Drive/Inputs/In/nState4 @bit 1 <-> WcState/InputToggle
//     Drive/Inputs/In/nState4 <-> WcState/WcState
//     Drive/Outputs/Out/nCtrl1 <-> DRV Controlword Channel 2/Controlword
//     Drive/Outputs/Out/nCtrl2 <-> DRV Controlword Channel 2/Controlword @bit 8
//     Drive/Outputs/Out/nDataOut1 <-> DRV Target position Channel 2/Target position
//     Enc/Inputs/In/nDataIn1 <-> FB Position Channel 2/Position
//     Enc/Inputs/In/nDcInputTime <-> InfoData/DcInputShift
//     Enc/Inputs/In/nState4 @bit 1 <-> WcState/InputToggle
//     Enc/Inputs/In/nState4 <-> WcState/WcState
//   NC-Task 1 SAF/Axes/Pump 7 - Linear <-> Device 3 (EtherCAT)/Term 22 (EK1100)/Term 29 (EL7062)
//     Drive/Inputs/In/nDataIn1 <-> DRV Following error actual value Channel 1/Following error actual value
//     Drive/Inputs/In/nDcOutputTime <-> InfoData/DcOutputShift
//     Drive/Inputs/In/nState1 <-> DRV Statusword Channel 1/Statusword
//     Drive/Inputs/In/nState2 <-> DRV Statusword Channel 1/Statusword @bit 8
//     Drive/Inputs/In/nState4 @bit 1 <-> WcState/InputToggle
//     Drive/Inputs/In/nState4 <-> WcState/WcState
//     Drive/Outputs/Out/nCtrl1 <-> DRV Controlword Channel 1/Controlword
//     Drive/Outputs/Out/nCtrl2 <-> DRV Controlword Channel 1/Controlword @bit 8
//     Drive/Outputs/Out/nDataOut1 <-> DRV Target position Channel 1/Target position
//     Enc/Inputs/In/nDataIn1 <-> FB Position Channel 1/Position
//     Enc/Inputs/In/nDcInputTime <-> InfoData/DcInputShift
//     Enc/Inputs/In/nState4 @bit 1 <-> WcState/InputToggle
//     Enc/Inputs/In/nState4 <-> WcState/WcState
//   NC-Task 1 SAF/Axes/Pump 7 - Rotary <-> Device 3 (EtherCAT)/Term 22 (EK1100)/Term 29 (EL7062)
//     Drive/Inputs/In/nDataIn1 <-> DRV Following error actual value Channel 2/Following error actual value
//     Drive/Inputs/In/nDcOutputTime <-> InfoData/DcOutputShift
//     Drive/Inputs/In/nState1 <-> DRV Statusword Channel 2/Statusword
//     Drive/Inputs/In/nState2 <-> DRV Statusword Channel 2/Statusword @bit 8
//     Drive/Inputs/In/nState4 @bit 1 <-> WcState/InputToggle
//     Drive/Inputs/In/nState4 <-> WcState/WcState
//     Drive/Outputs/Out/nCtrl1 <-> DRV Controlword Channel 2/Controlword
//     Drive/Outputs/Out/nCtrl2 <-> DRV Controlword Channel 2/Controlword @bit 8
//     Drive/Outputs/Out/nDataOut1 <-> DRV Target position Channel 2/Target position
//     Enc/Inputs/In/nDataIn1 <-> FB Position Channel 2/Position
//     Enc/Inputs/In/nDcInputTime <-> InfoData/DcInputShift
//     Enc/Inputs/In/nState4 @bit 1 <-> WcState/InputToggle
//     Enc/Inputs/In/nState4 <-> WcState/WcState
//   NC-Task 1 SAF/Axes/Pump 8 - Linear <-> Device 3 (EtherCAT)/Term 22 (EK1100)/Term 30 (EL7062)
//     Drive/Inputs/In/nDataIn1 <-> DRV Following error actual value Channel 1/Following error actual value
//     Drive/Inputs/In/nDcOutputTime <-> InfoData/DcOutputShift
//     Drive/Inputs/In/nState1 <-> DRV Statusword Channel 1/Statusword
//     Drive/Inputs/In/nState2 <-> DRV Statusword Channel 1/Statusword @bit 8
//     Drive/Inputs/In/nState4 @bit 1 <-> WcState/InputToggle
//     Drive/Inputs/In/nState4 <-> WcState/WcState
//     Drive/Outputs/Out/nCtrl1 <-> DRV Controlword Channel 1/Controlword
//     Drive/Outputs/Out/nCtrl2 <-> DRV Controlword Channel 1/Controlword @bit 8
//     Drive/Outputs/Out/nDataOut1 <-> DRV Target position Channel 1/Target position
//     Enc/Inputs/In/nDataIn1 <-> FB Position Channel 1/Position
//     Enc/Inputs/In/nDcInputTime <-> InfoData/DcInputShift
//     Enc/Inputs/In/nState4 @bit 1 <-> WcState/InputToggle
//     Enc/Inputs/In/nState4 <-> WcState/WcState
//   NC-Task 1 SAF/Axes/Pump 8 - Rotary <-> Device 3 (EtherCAT)/Term 22 (EK1100)/Term 30 (EL7062)
//     Drive/Inputs/In/nDataIn1 <-> DRV Following error actual value Channel 2/Following error actual value
//     Drive/Inputs/In/nDcOutputTime <-> InfoData/DcOutputShift
//     Drive/Inputs/In/nState1 <-> DRV Statusword Channel 2/Statusword
//     Drive/Inputs/In/nState2 <-> DRV Statusword Channel 2/Statusword @bit 8
//     Drive/Inputs/In/nState4 @bit 1 <-> WcState/InputToggle
//     Drive/Inputs/In/nState4 <-> WcState/WcState
//     Drive/Outputs/Out/nCtrl1 <-> DRV Controlword Channel 2/Controlword
//     Drive/Outputs/Out/nCtrl2 <-> DRV Controlword Channel 2/Controlword @bit 8
//     Drive/Outputs/Out/nDataOut1 <-> DRV Target position Channel 2/Target position
//     Enc/Inputs/In/nDataIn1 <-> FB Position Channel 2/Position
//     Enc/Inputs/In/nDcInputTime <-> InfoData/DcInputShift
//     Enc/Inputs/In/nState4 @bit 1 <-> WcState/InputToggle
//     Enc/Inputs/In/nState4 <-> WcState/WcState
//   NC-Task 1 SAF/Axes/Pump 9 - Linear <-> Device 3 (EtherCAT)/Term 22 (EK1100)/Term 31 (EL7062)
//     Drive/Inputs/In/nDataIn1 <-> DRV Following error actual value Channel 1/Following error actual value
//     Drive/Inputs/In/nDcOutputTime <-> InfoData/DcOutputShift
//     Drive/Inputs/In/nState1 <-> DRV Statusword Channel 1/Statusword
//     Drive/Inputs/In/nState2 <-> DRV Statusword Channel 1/Statusword @bit 8
//     Drive/Inputs/In/nState4 @bit 1 <-> WcState/InputToggle
//     Drive/Inputs/In/nState4 <-> WcState/WcState
//     Drive/Outputs/Out/nCtrl1 <-> DRV Controlword Channel 1/Controlword
//     Drive/Outputs/Out/nCtrl2 <-> DRV Controlword Channel 1/Controlword @bit 8
//     Drive/Outputs/Out/nDataOut1 <-> DRV Target position Channel 1/Target position
//     Enc/Inputs/In/nDataIn1 <-> FB Position Channel 1/Position
//     Enc/Inputs/In/nDcInputTime <-> InfoData/DcInputShift
//     Enc/Inputs/In/nState4 @bit 1 <-> WcState/InputToggle
//     Enc/Inputs/In/nState4 <-> WcState/WcState
//   NC-Task 1 SAF/Axes/Pump 9 - Rotary <-> Device 3 (EtherCAT)/Term 22 (EK1100)/Term 31 (EL7062)
//     Drive/Inputs/In/nDataIn1 <-> DRV Following error actual value Channel 2/Following error actual value
//     Drive/Inputs/In/nDcOutputTime <-> InfoData/DcOutputShift
//     Drive/Inputs/In/nState1 <-> DRV Statusword Channel 2/Statusword
//     Drive/Inputs/In/nState2 <-> DRV Statusword Channel 2/Statusword @bit 8
//     Drive/Inputs/In/nState4 @bit 1 <-> WcState/InputToggle
//     Drive/Inputs/In/nState4 <-> WcState/WcState
//     Drive/Outputs/Out/nCtrl1 <-> DRV Controlword Channel 2/Controlword
//     Drive/Outputs/Out/nCtrl2 <-> DRV Controlword Channel 2/Controlword @bit 8
//     Drive/Outputs/Out/nDataOut1 <-> DRV Target position Channel 2/Target position
//     Enc/Inputs/In/nDataIn1 <-> FB Position Channel 2/Position
//     Enc/Inputs/In/nDcInputTime <-> InfoData/DcInputShift
//     Enc/Inputs/In/nState4 @bit 1 <-> WcState/InputToggle
//     Enc/Inputs/In/nState4 <-> WcState/WcState
//   TE1063/TE1063 Instance <-> Device 3 (EtherCAT)/Box 1 (ifm IO-Link Master AL1333)
//     PlcTask Inputs/PRG_LevelHandler.byCh1_0 <-> Module 1 (IOL_In_4Byte)/TxPDO/input byte 0
//     PlcTask Inputs/PRG_LevelHandler.byCh1_1 <-> Module 1 (IOL_In_4Byte)/TxPDO/input byte 1
//     PlcTask Inputs/PRG_LevelHandler.byCh1_2 <-> Module 1 (IOL_In_4Byte)/TxPDO/input byte 2
//     PlcTask Inputs/PRG_LevelHandler.byCh1_3 <-> Module 1 (IOL_In_4Byte)/TxPDO/input byte 3
//     PlcTask Inputs/PRG_LevelHandler.byCh2_0 <-> Module 2 (IOL_In_4Byte)/TxPDO/input byte 0
//     PlcTask Inputs/PRG_LevelHandler.byCh2_1 <-> Module 2 (IOL_In_4Byte)/TxPDO/input byte 1
//     PlcTask Inputs/PRG_LevelHandler.byCh2_2 <-> Module 2 (IOL_In_4Byte)/TxPDO/input byte 2
//     PlcTask Inputs/PRG_LevelHandler.byCh2_3 <-> Module 2 (IOL_In_4Byte)/TxPDO/input byte 3
//     PlcTask Inputs/PRG_LevelHandler.byCh3_0 <-> Module 3 (IOL_In_4Byte)/TxPDO/input byte 0
//     PlcTask Inputs/PRG_LevelHandler.byCh3_1 <-> Module 3 (IOL_In_4Byte)/TxPDO/input byte 1
//     PlcTask Inputs/PRG_LevelHandler.byCh3_2 <-> Module 3 (IOL_In_4Byte)/TxPDO/input byte 2
//     PlcTask Inputs/PRG_LevelHandler.byCh3_3 <-> Module 3 (IOL_In_4Byte)/TxPDO/input byte 3
//     PlcTask Inputs/PRG_LevelHandler.byCh4_0 <-> Module 4 (IOL_In_4Byte)/TxPDO/input byte 0
//     PlcTask Inputs/PRG_LevelHandler.byCh4_1 <-> Module 4 (IOL_In_4Byte)/TxPDO/input byte 1
//     PlcTask Inputs/PRG_LevelHandler.byCh4_2 <-> Module 4 (IOL_In_4Byte)/TxPDO/input byte 2
//     PlcTask Inputs/PRG_LevelHandler.byCh4_3 <-> Module 4 (IOL_In_4Byte)/TxPDO/input byte 3
//     PlcTask Inputs/PRG_LevelHandler.byCh5_0 <-> Module 5 (IOL_In_4Byte)/TxPDO/input byte 0
//     PlcTask Inputs/PRG_LevelHandler.byCh5_1 <-> Module 5 (IOL_In_4Byte)/TxPDO/input byte 1
//     PlcTask Inputs/PRG_LevelHandler.byCh5_2 <-> Module 5 (IOL_In_4Byte)/TxPDO/input byte 2
//     PlcTask Inputs/PRG_LevelHandler.byCh5_3 <-> Module 5 (IOL_In_4Byte)/TxPDO/input byte 3
//     Task_Services Inputs/GVL_IO.nAL1333Box1State <-> InfoData/State
//     Task_Services Inputs/GVL_IO.stAL1333info.nQualifierIOLink[{1..8}] <-> TxPDO IO-Link Port Qualifier/Qualifier of IO-Link Ch.{1..8}  (8 links)
//     Task_Services Inputs/GVL_IO.stAL1333info.nStateIOLink[{1..8}] <-> TxPDO IO-Link Device Status/State of IO-Link Ch.{1..8}  (8 links)
//   TE1063/TE1063 Instance <-> Device 3 (EtherCAT)/Term 1 (EK1100)
//     Task_Services Inputs/GVL_IO.nEK1100T01State <-> InfoData/State
//   TE1063/TE1063 Instance <-> Device 3 (EtherCAT)/Term 1 (EK1100)/Term 10 (EL2809-0015)
//     PlcTask Outputs/GVL_IO.gDigOutputs/bResetIndicator <-> Channel 2/Output
//     PlcTask Outputs/GVL_IO.gDigOutputs/bSolenoidValveA <-> Channel 8/Output
//     PlcTask Outputs/GVL_IO.gDigOutputs/bSolenoidValveB <-> Channel 7/Output
//     PlcTask Outputs/GVL_IO.gDigOutputs/bSolenoidValveC <-> Channel 9/Output
//     PlcTask Outputs/GVL_IO.gDigOutputs/bStartIndicator <-> Channel 1/Output
//     PlcTask Outputs/GVL_IO.gDigOutputs/bTowerAmberLight <-> Channel 4/Output
//     PlcTask Outputs/GVL_IO.gDigOutputs/bTowerBuzzer <-> Channel 6/Output
//     PlcTask Outputs/GVL_IO.gDigOutputs/bTowerGreenLight <-> Channel 5/Output
//     PlcTask Outputs/GVL_IO.gDigOutputs/bTowerRedLight <-> Channel 3/Output
//     Task_Services Inputs/GVL_IO.nEL2809T10State <-> InfoData/State
//   TE1063/TE1063 Instance <-> Device 3 (EtherCAT)/Term 1 (EK1100)/Term 11 (EL2624)
//     PlcTask Outputs/GVL_IO.gRelayOutputs/bSampleRecoveryLight <-> Channel 2/Output
//     PlcTask Outputs/GVL_IO.gRelayOutputs/bStageCollectionLeftLight <-> Channel 1/Output
//     PlcTask Outputs/GVL_IO.gRelayOutputs/bStageCollectionRightLight <-> Channel 3/Output
//     Task_Services Inputs/GVL_IO.nEL2624T11State <-> InfoData/State
//   TE1063/TE1063 Instance <-> Device 3 (EtherCAT)/Term 1 (EK1100)/Term 12 (EL9410)
//     PlcTask Inputs/GVL_IO.bEL9410UPStatus <-> Status Up/Undervoltage
//     PlcTask Inputs/GVL_IO.bEL9410USStatus <-> Status Us/Undervoltage
//     Task_Services Inputs/GVL_IO.nEL9410T12State <-> InfoData/State
//   TE1063/TE1063 Instance <-> Device 3 (EtherCAT)/Term 1 (EK1100)/Term 13 (EL3058)
//     PlcTask Inputs/GVL_IO.gAnalogInputs/bLeakTestSensorError <-> AI Standard Channel 2/Status/Error
//     PlcTask Inputs/GVL_IO.gAnalogInputs/bMainPressureSupplyError <-> AI Standard Channel 1/Status/Error
//     PlcTask Inputs/GVL_IO.gAnalogInputs/bPressureRegulatorError <-> AI Standard Channel 3/Status/Error
//     PlcTask Inputs/GVL_IO.gAnalogInputs/rLeakTestPressureSensor <-> AI Standard Channel 2/Value
//     PlcTask Inputs/GVL_IO.gAnalogInputs/rMainPressureSupplyInput <-> AI Standard Channel 1/Value
//     PlcTask Inputs/GVL_IO.gAnalogInputs/rPressureRegulatorInput <-> AI Standard Channel 3/Value
//     Task_Services Inputs/GVL_IO.nEL3058T13State <-> InfoData/State
//   TE1063/TE1063 Instance <-> Device 3 (EtherCAT)/Term 1 (EK1100)/Term 14 (EL9576)
//     PlcTask Inputs/GVL_IO.bEL9576T14ChopperOn <-> BCT Inputs/Chopper on
//     PlcTask Inputs/GVL_IO.bEL9576T14DCLinkVoltage <-> BCT Inputs/DC link voltage
//     PlcTask Inputs/GVL_IO.bEL9576T14I2TError <-> BCT Inputs/I2T error
//     PlcTask Inputs/GVL_IO.bEL9576T14I2TWarning <-> BCT Inputs/I2T warning
//     PlcTask Inputs/GVL_IO.bEL9576T14OverCurrent <-> BCT Inputs/Overcurrent Protection
//     PlcTask Inputs/GVL_IO.bEL9576T14OverVoltage <-> BCT Inputs/Overvoltage
//     PlcTask Inputs/GVL_IO.bEL9576T14Overtemp <-> BCT Inputs/Terminal Overtemperature
//     PlcTask Inputs/GVL_IO.bEL9576T14UnderVoltage <-> BCT Inputs/Undervoltage
//     Task_Services Inputs/GVL_IO.nEL9576T14State <-> InfoData/State
//   TE1063/TE1063 Instance <-> Device 3 (EtherCAT)/Term 1 (EK1100)/Term 15 (EL7211-9014)
//     PlcTask Inputs/GVL_Motion.M2Motor.nState <-> InfoData/State
//   TE1063/TE1063 Instance <-> Device 3 (EtherCAT)/Term 1 (EK1100)/Term 16 (EL7211-9014)
//     PlcTask Inputs/GVL_Motion.M3Motor.nState <-> InfoData/State
//   TE1063/TE1063 Instance <-> Device 3 (EtherCAT)/Term 1 (EK1100)/Term 17 (EL3022)
//     PlcTask Inputs/GVL_IO.bEL3022ChAError <-> AI Standard Channel 1/Error
//     PlcTask Inputs/GVL_IO.bEL3022ChAOverRange <-> AI Standard Channel 1/Overrange
//     PlcTask Inputs/GVL_IO.bEL3022ChAUnderRange <-> AI Standard Channel 1/Underrange
//     PlcTask Inputs/GVL_IO.bEL3022ChBError <-> AI Standard Channel 2/Error
//     PlcTask Inputs/GVL_IO.bEL3022ChBOverRange <-> AI Standard Channel 2/Overrange
//     PlcTask Inputs/GVL_IO.bEL3022ChBUnderRange <-> AI Standard Channel 2/Underrange
//     Task_Services Inputs/GVL_IO.nEL3022T17State <-> InfoData/State
//   TE1063/TE1063 Instance <-> Device 3 (EtherCAT)/Term 1 (EK1100)/Term 18 (EL1809)
//     PlcTask Inputs/GVL_IO.gDigInputs/bAccessDoor4InterlockFdbk <-> Channel 1/Input
//     PlcTask Inputs/GVL_IO.gDigInputs/bAccessDoor5InterlockFdbk <-> Channel 2/Input
//     PlcTask Inputs/GVL_IO.gDigInputs/bAccessDoor6InterlockFdbk <-> Channel 3/Input
//     Task_Services Inputs/GVL_IO.nEL1809T18State <-> InfoData/State
//   TE1063/TE1063 Instance <-> Device 3 (EtherCAT)/Term 1 (EK1100)/Term 19 (EL2904)
//     PlcTask Inputs/GVL_IO.nEL2904T19State <-> InfoData/State
//   TE1063/TE1063 Instance <-> Device 3 (EtherCAT)/Term 1 (EK1100)/Term 2 (EL6070-0033)
//     Task_Services Inputs/GVL_IO.nEL6070State <-> InfoData/State
//   TE1063/TE1063 Instance <-> Device 3 (EtherCAT)/Term 1 (EK1100)/Term 20 (EL6631)
//     Task_Services Inputs/GVL_IO.nEL6631T20State <-> InfoData/State
//   TE1063/TE1063 Instance <-> Device 3 (EtherCAT)/Term 1 (EK1100)/Term 3 (EL6910)
//     PlcTask Inputs/GVL_IO.stEL6910.nEL6910State <-> InfoData/State
//     PlcTask Inputs/GVL_Safety.SafetyInputs/bM1STOEnabled <-> StandardInputs/Standard Out Var 22
//     PlcTask Inputs/GVL_Safety.SafetyInputs/bSafetyAirError <-> StandardInputs/Standard Out Var 16
//     PlcTask Inputs/GVL_Safety.SafetyInputs/bSafetyAirPressurising <-> StandardInputs/Standard Out Var 20
//     PlcTask Inputs/GVL_Safety.SafetyInputs/iSafetyEStop <-> StandardInputs/Standard Out Var 21
//     PlcTask Inputs/GVL_Safety.aEL2904_T07[1] <-> StandardInputs/Standard Out Var 116
//     PlcTask Inputs/GVL_Safety.aEL2904_T07[2] <-> StandardInputs/Standard Out Var 117
//     PlcTask Inputs/GVL_Safety.aEL2904_T07[3] <-> StandardInputs/Standard Out Var 118
//     PlcTask Inputs/GVL_Safety.aEL2904_T08[1] <-> StandardInputs/Standard Out Var 119
//     PlcTask Inputs/GVL_Safety.aEL2904_T08[2] <-> StandardInputs/Standard Out Var 120
//     PlcTask Inputs/GVL_Safety.aEL2904_T08[3] <-> StandardInputs/Standard Out Var 121
//     PlcTask Inputs/GVL_Safety.aEL2904_T08[4] <-> StandardInputs/Standard Out Var 122
//     PlcTask Inputs/GVL_Safety.aEL2904_T19[1] <-> StandardInputs/Standard Out Var 123
//     PlcTask Inputs/GVL_Safety.aEL2904_T19[2] <-> StandardInputs/Standard Out Var 124
//     PlcTask Inputs/GVL_Safety.aEL2904_T19[3] <-> StandardInputs/Standard Out Var 125
//     PlcTask Inputs/GVL_Safety.bDoorClosedAlias <-> StandardInputs/Standard Out Var 17
//     PlcTask Inputs/GVL_Safety.bDoorLockedFeedback <-> StandardInputs/Standard Out Var 13
//     PlcTask Inputs/GVL_Safety.bM1STOEnabled <-> StandardInputs/Standard Out Var 25
//     PlcTask Inputs/GVL_Safety.bM1STOErrorAck <-> StandardInputs/Standard Out Var 44
//     PlcTask Inputs/GVL_Safety.bResetButtonBlink <-> StandardInputs/Standard Out Var 95
//     PlcTask Inputs/GVL_Safety.bSafetyEnable <-> StandardInputs/Standard Out Var 97
//     PlcTask Inputs/GVL_Safety.iMotorsSTOEnabled <-> StandardInputs/Standard Out Var 73
//     PlcTask Outputs/GVL_Safety.SafetyOutputs/bAirPressureOK <-> StandardOutputs/Standard In Var 14
//     PlcTask Outputs/GVL_Safety.SafetyOutputs/bBelowDoorsFeedback <-> StandardOutputs/Standard In Var 43
//     PlcTask Outputs/GVL_Safety.SafetyOutputs/bResetAir <-> StandardOutputs/Standard In Var 15
//     PlcTask Outputs/GVL_Safety.bAirSupplyEnable <-> StandardOutputs/Standard In Var 93
//     PlcTask Outputs/GVL_Safety.bAirSupplyReset <-> StandardOutputs/Standard In Var 94
//     PlcTask Outputs/GVL_Safety.bDoor3BypassAccepted <-> StandardOutputs/Standard In Var 112
//     PlcTask Outputs/GVL_Safety.bDoorLockCommand <-> StandardOutputs/Standard In Var 12
//     PlcTask Outputs/GVL_Safety.bImmediateFaultCommand <-> StandardOutputs/Standard In Var 126
//     PlcTask Outputs/GVL_Safety.bSafetyErrorAck <-> StandardOutputs/Standard In Var 7
//     PlcTask Outputs/GVL_Safety.bSafetyRun <-> StandardOutputs/Standard In Var 8
//     Task_Services Inputs/GVL_IO.stEL6910.iSafetyComError <-> StandardInputs/Standard Out Var 113
//     Task_Services Inputs/GVL_IO.stEL6910.iSafetyFBError <-> StandardInputs/Standard Out Var 114
//     Task_Services Inputs/GVL_IO.stEL6910.iSafetyRunning <-> StandardInputs/Standard Out Var 115
//     Task_Services Inputs/GVL_Safety.bAirEnabledFeedback <-> StandardInputs/Standard Out Var 18
//     Task_Services Inputs/GVL_Safety.bTopDoorsClosedFeedback <-> StandardInputs/Standard Out Var 110
//     Task_Services Outputs/GVL_Safety.bSafetyRestart <-> StandardOutputs/Standard In Var 9
//   TE1063/TE1063 Instance <-> Device 3 (EtherCAT)/Term 1 (EK1100)/Term 4 (EL1918)
//     PlcTask Inputs/GVL_IO.nEL1918T04State <-> InfoData/State
//     PlcTask Inputs/GVL_Safety.SafetyInputs/bEStopHMICh1 <-> Module 1 (FSOE)/FSoE Inputs/FSOE/FSIN Module 1.Input
//     PlcTask Inputs/GVL_Safety.SafetyInputs/bEStopHMICh2 <-> Module 1 (FSOE)/FSoE Inputs/FSOE/FSIN Module 2.Input
//     PlcTask Inputs/GVL_Safety.SafetyInputs/bEStopSideCh1 <-> Module 1 (FSOE)/FSoE Inputs/FSOE/FSIN Module 3.Input
//     PlcTask Inputs/GVL_Safety.SafetyInputs/bEStopSideCh2 <-> Module 1 (FSOE)/FSoE Inputs/FSOE/FSIN Module 4.Input
//     PlcTask Inputs/GVL_Safety.SafetyInputs/bMachineReset <-> Module 1 (FSOE)/FSoE Inputs/FSOE/FSIN Module 5.Input
//     PlcTask Inputs/GVL_Safety.SafetyInputs/bStageCollectLeftDoorCh1 <-> Module 1 (FSOE)/FSoE Inputs/FSOE/FSIN Module 6.Input
//     PlcTask Inputs/GVL_Safety.SafetyInputs/bStageCollectLeftDoorCh2 <-> Module 1 (FSOE)/FSoE Inputs/FSOE/FSIN Module 7.Input
//     PlcTask Inputs/GVL_Safety.SafetyInputs/bStageCollectLeftDoorFdbk <-> Module 1 (FSOE)/FSoE Inputs/FSOE/FSIN Module 8.Input
//   TE1063/TE1063 Instance <-> Device 3 (EtherCAT)/Term 1 (EK1100)/Term 5 (EL1918)
//     PlcTask Inputs/GVL_IO.nEL1918T05State <-> InfoData/State
//     PlcTask Inputs/GVL_Safety.SafetyInputs/bSampleRecoveryDoorCh1 <-> Module 1 (FSOE)/FSoE Inputs/FSOE/FSIN Module 4.Input
//     PlcTask Inputs/GVL_Safety.SafetyInputs/bSampleRecoveryDoorCh2 <-> Module 1 (FSOE)/FSoE Inputs/FSOE/FSIN Module 5.Input
//     PlcTask Inputs/GVL_Safety.SafetyInputs/bSampleRecoveryDoorFdbk <-> Module 1 (FSOE)/FSoE Inputs/FSOE/FSIN Module 6.Input
